//前破壞電磁閥
F_TRIG_2(CLK:=SOL_S8_VacuumF);
interlockback[3]:=TRUE;
interlockout[3]:=TRUE;
(*SET*)
IF ((F_TRIG_2.Q AND NOT(solstatus[3]))) AND interlockout[3] THEN
	SOL_S8_BreakF:=TRUE;
END_IF;
(*RESET*)
TON_BreakF(In:=SOL_S8_BreakF, PT:=t#500ms);
IF ((TON_BreakF.Q AND (solstatus[3]))) AND interlockback[3] THEN
	SOL_S8_BreakF:=FALSE;
END_IF;
(*STATUS*)
solstatus[3]:=SOL_S8_BreakF;

//後吸取電磁閥
R_TRIG_1[4](CLK:=HMIPB_SOL_S8_VacuumR AND NOT(AutoStatus));
interlockback[4]:=TRUE;
interlockout[4]:=TRUE;
(*SET*)
IF ((R_TRIG_1[4].Q AND NOT(solstatus[4])) OR Autoflow=3) AND interlockout[4] THEN
	SOL_S8_VacuumR:=TRUE;
END_IF;
(*RESET*)
IF ((R_TRIG_1[4].Q AND (solstatus[4])) OR Autoflow=7 OR Initflow=7 OR ErrorStatus[8]) AND interlockback[4] THEN
	SOL_S8_VacuumR:=FALSE;
END_IF;
(*STATUS*)
solstatus[4]:=SOL_S8_VacuumR;

//後破壞電磁閥
F_TRIG_3(CLK:=SOL_S8_VacuumR);
interlockback[5]:=TRUE;
interlockout[5]:=TRUE;
(*SET*)
IF ((F_TRIG_3.Q AND NOT(solstatus[5]))) AND interlockout[5] THEN
	SOL_S8_BreakR:=TRUE;
END_IF;
(*RESET*)
TON_BreakR(In:=SOL_S8_BreakR, PT:=t#500ms);
IF ((TON_BreakR.Q AND (solstatus[5]))) AND interlockback[5] THEN
	SOL_S8_BreakR:=FALSE;
END_IF;
(*STATUS*)
solstatus[5]:=SOL_S8_BreakR;
(*************************************************************************
程序名稱:第8站卡子RESET流程
作者:蔡相偉
版本,日期,版本資訊:
1.0.0		2017/11/22		初始版本

PowerOn=0
Idle=1
夾取回=7
上下回=8
移位回=9
*************************************************************************)
//PowerOn=0
IF NOT(SystemReadyStatus) THEN
	Initflow:=0;
END_IF;

//Idle=1
IF Initflow=0 AND SystemReadyStatus THEN
	Initflow:=1;
END_IF;

IF Initflow=9 AND LS_S8_MoveBack THEN
	Initflow:=1;
END_IF;

//夾取回=7
F_TRIG_1(CLK:= ErrorStatus[8] OR Error_PB_Estop);
IF Initflow=1 AND (F_TRIG_1.Q OR Manual2AutoFlag) THEN
	Initflow:=7;
END_IF;

//上下回=8
IF Initflow=7 AND NOT(SOL_S8_VacuumF) AND NOT(SNR_S8_VacuumF) AND NOT(SOL_S8_VacuumR) AND NOT(SNR_S8_VacuumR) THEN
	Initflow:=8;
END_IF;

//移位回=9
IF Initflow=8 AND LS_S8_UpDownBack THEN
	Initflow:=9;
END_IF;

//*************************************************************************
//Cycle Time
//*************************************************************************
TON_CT(In:=AutoFlow>1, PT:=t#500s);
IF Autoflow>1 THEN
CycleTime[8]:=LINT_TO_REAL(TimeToNanoSec( TON_CT.ET))/1000000000.0;
END_IF;
END_PROGRAM

PROGRAM prStation8_CCD
VAR
    Autoflow : INT;
    R_TRIG_1 : R_TRIG;
    F_TRIG_1 : F_TRIG;
END_VAR
VAR_EXTERNAL
    SystemReadyStatus : BOOL;
    AutoStatus : BOOL;
    HMIPB_OMRON_FQ2_Trig : BOOL;
    OMRON_FQ2_Trig : BOOL;
    OMRON_FQ2_IN0 : BOOL;
    OMRON_FQ2_IN1 : BOOL;
    OMRON_FQ2_IN2 : BOOL;
    OMRON_FQ2_IN3 : BOOL;
    OMRON_FQ2_IN4 : BOOL;
    OMRON_FQ2_IN5 : BOOL;
    CCD_Check_NG : BOOL;
    OMRON_FQ2_Ready : BOOL;
    OMRON_FQ2_NG : BOOL;
    CCDStartFlag : BOOL;
    CCDFinishFlag : BOOL;
END_VAR
(*************************************************************************
程序名稱:CCD流程
作者:蔡相偉
版本,日期,版本資訊:
1.0.0	2016/6/3		初始版本,SNR感測到立即拍照
2.0.0	2016/10/11		修改在轉盤站上使用
流程
PowerOn=0
Idle=1
工件到位=5
CCD拍攝中=2
CCD拍攝完成=3
CCD判定資料記錄=4
工件離開=6
*************************************************************************)
//PowerOn=0
IF NOT(SystemReadyStatus AND AutoStatus) THEN
	AutoFlow:=0;
END_IF;

(*Idle=1*)
IF AutoFlow=0 AND SystemReadyStatus AND AutoStatus THEN
	AutoFlow:=1;
END_IF;

IF AutoFlow=6 AND NOT(CCDStartFlag) THEN
	AutoFlow:=1;
END_IF;

(*工件到位=5*)
IF Autoflow=1 AND CCDStartFlag THEN
	Autoflow:=5;
	CCD_Check_NG:=FALSE;
END_IF;

(*CCD拍攝中=2*)
IF AutoFlow=5  AND OMRON_FQ2_Ready THEN
	AutoFlow:=2;
END_IF;

(*CCD拍攝完成=3*)
IF AutoFlow=2 AND NOT(OMRON_FQ2_Ready) THEN
	AutoFlow:=3;
END_IF;

(*CCD判定資料記錄=4*)
IF AutoFlow=3 THEN
	AutoFlow:=4;
END_IF;

(*工件離開=6*)
IF AutoFlow=4 THEN
	IF OMRON_FQ2_NG THEN
		CCD_Check_NG:=TRUE;
	END_IF;
	AutoFlow:=6;
END_IF;
IF Autoflow=6 THEN
	CCDFinishFlag:=TRUE;
ELSE
	CCDFinishFlag:=FALSE;
END_IF;

//****************************************************************************************
(*手動*)
R_TRIG_1(CLK:= HMIPB_OMRON_FQ2_Trig);
IF R_TRIG_1.Q OR AutoFlow=5 THEN
	OMRON_FQ2_Trig:=TRUE;
END_IF;
F_TRIG_1(CLK:= HMIPB_OMRON_FQ2_Trig);
IF F_TRIG_1.Q OR AutoFlow=2 THEN
	OMRON_FQ2_Trig:=FALSE;
END_IF;

(*場景選擇*)
OMRON_FQ2_IN0:=FALSE;
OMRON_FQ2_IN1:=FALSE;
OMRON_FQ2_IN2:=FALSE;
OMRON_FQ2_IN3:=FALSE;
OMRON_FQ2_IN4:=FALSE;
OMRON_FQ2_IN5:=FALSE;
END_PROGRAM

PROGRAM prStation8_ChangeJig
VAR
    interlockback : ARRAY[0..5] OF BOOL;
    interlockout : ARRAY[0..5] OF BOOL;
    R_TRIG_1 : ARRAY[0..5] OF R_TRIG;
    solstatus : ARRAY[0..5] OF BOOL;
    Autoflow : INT;
    Initflow : INT;
    F_TRIG_1 : F_TRIG;
    Rtrig_test : R_TRIG;
    TON1 : TON;
END_VAR
VAR_EXTERNAL
    HMIPB_SOL_S8_Fix : BOOL;
    AutoStatus : BOOL;
    SOL_S8_Fix : BOOL;
    HMIPB_SOL_S8_FixMove : BOOL;
    SOL_S8_FixMove : BOOL;
    HMIPB_SOL_S8_Turn : BOOL;
    SOL_S8_Turn : BOOL;
    HMIPB_SOL_S8_Clip : BOOL;
    SOL_S8_Clip : BOOL;
    SystemReadyStatus : BOOL;
    CCDStartFlag : BOOL;
    CCD_Check_NG : BOOL;
    S8_ChangeJigStartFlag : BOOL;
    LS_S8_FixMoveOut : BOOL;
    ErrorStatus_S8_Fix : BOOL;
    LS_S8_ClipOut : BOOL;
    LS_S8_FixOut : BOOL;
    LS_S8_TurnOut : BOOL;
    LS_S8_FixBack : BOOL;
    LS_S8_ClipBack : BOOL;
    LS_S8_FixMoveBack : BOOL;
    LS_S8_TurnBack : BOOL;
    LS_S8_MoveBack : BOOL;
    ErrorStatus : ARRAY[0..19] OF BOOL;
    Error_PB_EStop : BOOL;
    Manual2AutoFlag : BOOL;
    StepMode : BOOL;
    LS_S8_UpDownBack : BOOL;
    SOL_S8_UpDown : BOOL;
END_VAR
(*************************************************************************
程序名稱:換卡子方向流程
作者:蔡相偉
版本,日期,版本資訊:
1.0.0		2017/11/29		初始版本

PowerOn=0
Idle=1
前後出=2
夾取出=3
定位出=4
旋轉出=5
定位回=6
夾取回=7
前後回=8
旋轉回=9
*************************************************************************)
//PowerOn=0
IF NOT(SystemReadyStatus AND AutoStatus AND NOT(ErrorStatus_S8_Fix)) THEN
	AutoFlow:=0;
END_IF;

(*Idle=1*)
IF AutoFlow=0 AND SystemReadyStatus AND AutoStatus AND NOT(ErrorStatus_S8_Fix) THEN
	AutoFlow:=1;
END_IF;

IF AutoFlow=9 AND LS_S8_TurnBack THEN
	AutoFlow:=1;
END_IF;

//前後出=2
IF Autoflow=1 AND S8_ChangeJigStartFlag AND Initflow=1 THEN
	Autoflow:=2;
END_IF;

//夾取出=3
IF Autoflow=2 AND LS_S8_FixMoveOut AND (Rtrig_test.Q OR NOT(StepMode)) THEN
	Autoflow:=3;
END_IF;

//定位出=4
IF Autoflow=3 AND LS_S8_ClipOut AND (Rtrig_test.Q OR NOT(StepMode)) THEN
	Autoflow:=4;
END_IF;

//旋轉出=5
IF Autoflow=4 AND LS_S8_FixOut AND (Rtrig_test.Q OR NOT(StepMode)) THEN
	Autoflow:=5;
END_IF;
TON1(In:=Autoflow=5 AND LS_S8_TurnOut, PT:=t#300ms);
//定位回=6
IF Autoflow=5 AND TON1.Q AND (Rtrig_test.Q OR NOT(StepMode)) THEN
	Autoflow:=6;
	S8_ChangeJigStartFlag:=FALSE;
END_IF;

//夾取回=7
IF Autoflow=6 AND LS_S8_FixBack AND (Rtrig_test.Q OR NOT(StepMode)) THEN
	Autoflow:=7;
END_IF;

//前後回=8
IF Autoflow=7 AND LS_S8_ClipBack AND (Rtrig_test.Q OR NOT(StepMode)) THEN
	Autoflow:=8;
END_IF;

//旋轉回=9
IF Autoflow=8 AND LS_S8_FixMoveBack AND (Rtrig_test.Q OR NOT(StepMode)) THEN
	Autoflow:=9;
END_IF;

//*************************************************************************
//手動
//定位電磁閥
R_TRIG_1[0](CLK:=HMIPB_SOL_S8_Fix AND NOT(AutoStatus));
interlockback[0]:=TRUE;
interlockout[0]:=TRUE;
(*SET*)
IF ((R_TRIG_1[0].Q AND NOT(solstatus[0])) OR Autoflow=4) AND interlockout[0] THEN
	SOL_S8_Fix:=TRUE;
END_IF;
(*RESET*)
IF ((R_TRIG_1[0].Q AND (solstatus[0])) OR Autoflow=6 OR Initflow=6) AND interlockback[0] THEN
	SOL_S8_Fix:=FALSE;
END_IF;
(*STATUS*)
solstatus[0]:=SOL_S8_Fix;

//定位前後電磁閥
R_TRIG_1[1](CLK:=HMIPB_SOL_S8_FixMove AND NOT(AutoStatus));
interlockback[1]:=TRUE;
interlockout[1]:=TRUE;
(*SET*)
IF ((R_TRIG_1[1].Q AND NOT(solstatus[1])) OR Autoflow=2) AND interlockout[1] THEN
	SOL_S8_FixMove:=TRUE;
END_IF;
(*RESET*)
IF ((R_TRIG_1[1].Q AND (solstatus[1])) OR Autoflow=8 OR Initflow=8) AND interlockback[1] THEN
	SOL_S8_FixMove:=FALSE;
END_IF;
(*STATUS*)
solstatus[1]:=SOL_S8_FixMove;

//定位旋轉電磁閥
R_TRIG_1[2](CLK:=HMIPB_SOL_S8_Turn AND NOT(AutoStatus));
interlockback[2]:=(LS_S8_FixOut AND SOL_S8_Fix AND LS_S8_UpDownBack AND NOT(SOL_S8_UpDown)) OR LS_S8_FixMoveBack;
interlockout[2]:=(LS_S8_FixOut AND SOL_S8_Fix AND LS_S8_UpDownBack AND NOT(SOL_S8_UpDown)) OR LS_S8_FixMoveBack;
(*SET*)
IF ((R_TRIG_1[2].Q AND NOT(solstatus[2])) OR Autoflow=5) AND interlockout[2] THEN
	SOL_S8_Turn:=TRUE;
END_IF;
(*RESET*)
IF ((R_TRIG_1[2].Q AND (solstatus[2])) OR Autoflow=9 OR Initflow=9) AND interlockback[2] THEN
	SOL_S8_Turn:=FALSE;
END_IF;
(*STATUS*)
solstatus[2]:=SOL_S8_Turn;

//定位夾持電磁閥
R_TRIG_1[3](CLK:=HMIPB_SOL_S8_Clip AND NOT(AutoStatus));
interlockback[3]:=TRUE;
interlockout[3]:=TRUE;
(*SET*)
IF ((R_TRIG_1[3].Q AND NOT(solstatus[3])) OR Autoflow=3) AND interlockout[3] THEN
	SOL_S8_Clip:=TRUE;
END_IF;
(*RESET*)
IF ((R_TRIG_1[3].Q AND (solstatus[3])) OR Autoflow=7 OR Initflow=7) AND interlockback[3] THEN
	SOL_S8_Clip:=FALSE;
END_IF;
(*STATUS*)
solstatus[3]:=SOL_S8_Clip;
(*************************************************************************
程序名稱:換卡子方向RESET流程
作者:蔡相偉
版本,日期,版本資訊:
1.0.0		2017/11/29		初始版本

PowerOn=0
Idle=1
定位回=6
夾取回=7
前後回=8
旋轉回=9
*************************************************************************)
//PowerOn=0
IF NOT(SystemReadyStatus) THEN
	Initflow:=0;
END_IF;

//Idle=1
IF Initflow=0 AND SystemReadyStatus THEN
	Initflow:=1;
END_IF;

IF Initflow=9 AND LS_S8_TurnBack THEN
	Initflow:=1;
END_IF;

//定位回=6
F_TRIG_1(CLK:= ErrorStatus_S8_Fix);
IF Initflow=1 AND (F_TRIG_1.Q) THEN
	Initflow:=6;
END_IF;

//夾取回=7
IF Initflow=6 AND LS_S8_FixBack THEN
	Initflow:=7;
END_IF;

//前後回=8
IF Initflow=7 AND LS_S8_ClipBack THEN
	Initflow:=8;
END_IF;

//旋轉回=9
IF Initflow=8 AND LS_S8_FixMoveBack THEN
	Initflow:=9;
END_IF;
END_PROGRAM

PROGRAM prStation9
VAR
    interlockback : ARRAY[0..1] OF BOOL;
    interlockout : ARRAY[0..1] OF BOOL;
    solstatus : ARRAY[0..1] OF BOOL;
    R_TRIG_1 : ARRAY[0..1] OF R_TRIG;
    Rtrig_test : R_TRIG;
    F_TRIG_1 : F_TRIG;
    Autoflow : INT;
    Initflow : INT;
    TON1 : TON;
    TON2 : TON;
    TON_CT : TON;
END_VAR
VAR_EXTERNAL
    IndexData : ARRAY[0..19] OF stIndexData;
    DisablePB : ARRAY[0..19] OF BOOL;
    SystemReadyStatus : BOOL;
    AutoStatus : BOOL;
    ErrorStatus : ARRAY[0..19] OF BOOL;
    Error_PB_EStop : BOOL;
    MachineRunStatus : BOOL;
    SNR_Index : BOOL;
    RY_Index : BOOL;
    Manual2AutoFlag : BOOL;
    TestPB : ARRAY[0..19] OF BOOL;
    SNR_S9_Check : BOOL;
    CycleTime : ARRAY[0..19] OF REAL;
    BatchIndexCount : DINT;
    Error_SNR_S9_Check : BOOL;
    PB_Reset : BOOL;
    HMIPB_PB_Reset : BOOL;
    Error_SNR_S5_Check : BOOL;
    BatchNGCount : DINT;
END_VAR
(*************************************************************************
程序名稱:第9站檢查卡子流程
作者:蔡相偉
版本,日期,版本資訊:
1.0.0		2017/11/22		初始版本

PowerOn=0
Idle=1
檢查開始=2
檢查完成=3
*************************************************************************)
(*************************************************************************
異常碼
急停=1
氣缸=2
檢查NG=3
*************************************************************************)
//*************************************************************************
//本站狀態判斷
IF IndexData[9].OKFlag[9]
	OR IndexData[9].NGFlag[9] THEN
	IndexData[9].FinishFlag[9]:=TRUE;
END_IF;
//前站狀態判斷
IF  NOT(IndexData[9].FinishFlag[8]) OR	IndexData[9].NGFlag[8] THEN
	IndexData[9].NGFlag[9]:=TRUE;
END_IF;
//本站關閉判斷
IF DisablePB[9] AND IndexData[9].FinishFlag[8] AND IndexData[9].OKFlag[8] AND NOT(IndexData[9].NGFlag[8]) THEN
	IndexData[9].OKFlag[9]:=TRUE;
END_IF;

Rtrig_test(CLK:=TestPB[9]);
//PowerOn=0
IF NOT(SystemReadyStatus AND AutoStatus AND NOT(ErrorStatus[9]) AND NOT(Error_PB_EStop)) THEN
	Autoflow:=0;
END_IF;
	//EStop異常碼
	(*IF Error_PB_Estop AND NOT(IndexData[4].FinishFlag[4]) AND IndexData[4].OkFlag[1] THEN
		IndexData[4].NGFlag[4]:=TRUE;
		IndexData[4].ErrorLog[4]:=1;
	END_IF;*)
	//Error異常碼
	(*IF ErrorStatus[4] AND NOT(IndexData[4].FinishFlag[4]) AND IndexData[4].OkFlag[1] THEN
		IndexData[4].NGFlag[4]:=TRUE;
		IndexData[4].ErrorLog[4]:=2;
	END_IF;*)
//Idle=1
IF AutoFlow=0 AND SystemReadyStatus AND AutoStatus AND NOT(ErrorStatus[9]) AND NOT(Error_PB_EStop) THEN
	AutoFlow:=1;
END_IF;

IF Autoflow=3 AND IndexData[9].FinishFlag[9] THEN
	Autoflow:=1;
END_IF;

//檢查開始=2
IF Autoflow=1
	AND AutoStatus
	AND NOT(DisablePB[9])
	AND SNR_Index
	AND NOT(RY_Index)
	AND (MachineRunStatus AND NOT(IndexData[9].FinishFlag[9]) AND IndexData[9].FinishFlag[8] AND IndexData[9].OKFlag[8] AND NOT(IndexData[9].NGFlag[8])
	OR Rtrig_test.Q) THEN
	Autoflow:=2;
	Error_SNR_S9_Check:=FALSE;
END_IF;
TON1(In:=Autoflow=2 AND SNR_S9_Check, PT:=t#500ms);		//OK
TON2(In:=Autoflow=2 AND NOT(TON1.Q), PT:=t#1000ms);		//NG
//檢查完成=3
IF Autoflow=2 AND TON1.Q THEN
	IndexData[9].OKFlag[9]:=TRUE;
	IndexData[9].NGFlag[9]:=FALSE;
	IndexData[9].ErrorLog[9]:=0;
	Autoflow:=3;
END_IF;
IF Autoflow=2 AND TON2.Q THEN
	Error_SNR_S9_Check:=TRUE;
	IndexData[9].OKFlag[9]:=FALSE;
	IndexData[9].NGFlag[9]:=TRUE;
	IndexData[9].ErrorLog[9]:=3;
	BatchIndexCount:=BatchIndexCount-1;
	BatchNGCount:=BatchNGCount+1;
	Autoflow:=3;
END_IF;
IF NOT(SNR_Index) THEN
	Error_SNR_S9_Check:=FALSE;
END_IF;
//*************************************************************************
//Cycle Time
//*************************************************************************
TON_CT(In:=AutoFlow>1, PT:=t#500s);
IF Autoflow>1 THEN
CycleTime[9]:=LINT_TO_REAL(TimeToNanoSec( TON_CT.ET))/1000000000.0;
END_IF;
END_PROGRAM

PROGRAM prStation10
VAR
    interlockback : ARRAY[0..4] OF BOOL;
    interlockout : ARRAY[0..4] OF BOOL;
    solstatus : ARRAY[0..4] OF BOOL;
    R_TRIG_1 : ARRAY[0..4] OF R_TRIG;
    Rtrig_test : R_TRIG;
    F_TRIG_1 : F_TRIG;
    Autoflow : INT;
    Initflow : INT;
    TON1 : TON;
    TON2 : TON;
    TON_CT : TON;
END_VAR
VAR_EXTERNAL
    HMIPB_SOL_S10_MoveBack : BOOL;
    AutoStatus : BOOL;
    SOL_S10_MoveBack : BOOL;
    SOL_S10_MoveOut : BOOL;
    LS_S10_MoveBack : BOOL;
    HMIPB_SOL_S10_MoveOut : BOOL;
    LS_S10_MoveOut : BOOL;
    HMIPB_SOL_S10_UpDown : BOOL;
    SOL_S10_UpDown : BOOL;
    IndexData : ARRAY[0..19] OF stIndexData;
    DisablePB : ARRAY[0..19] OF BOOL;
    TestPB : ARRAY[0..19] OF BOOL;
    SystemReadyStatus : BOOL;
    ErrorStatus : ARRAY[0..19] OF BOOL;
    Error_PB_EStop : BOOL;
    Error_SNR_S10_Feed : BOOL;
    LS_S10_UpDownBack : BOOL;
    MachineRunStatus : BOOL;
    LS_S10_UpDownOut : BOOL;
    SNR_Index : BOOL;
    RY_Index : BOOL;
    Manual2AutoFlag : BOOL;
    YAMAHA_ORG : BOOL;
    SNR_S10_Feed : BOOL;
    FeedStart : ARRAY[0..19] OF BOOL;
    FeedFinish : ARRAY[0..19] OF BOOL;
    ErrorStatus_TH : ARRAY[0..19] OF BOOL;
    LS_S2_UpDownOut : BOOL;
    HMIPB_SOL_S10_ClipF : BOOL;
    SOL_S10_ClipF : BOOL;
    HMIPB_SOL_S10_ClipR : BOOL;
    SOL_S10_ClipR : BOOL;
    HMIPB_SOL_S10_Turn : BOOL;
    SOL_S10_Turn : BOOL;
    LS_S10_THBack : BOOL;
    LS_S10_ClipFBack : BOOL;
    LS_S10_ClipRBack : BOOL;
    LS_S10_TurnBack : BOOL;
    LS_S10_ClipFOut : BOOL;
    LS_S10_ClipROut : BOOL;
    LS_S10_TurnOut : BOOL;
    CycleTime : ARRAY[0..19] OF REAL;
    BatchIndexCount : DINT;
    Error_LS_S10_UpDownOut1 : BOOL;
    StepMode : BOOL;
    BatchNGCount : DINT;
END_VAR
(*************************************************************************
程序名稱:第10站上夾板流程
作者:蔡相偉
版本,日期,版本資訊:
1.0.0		2017/11/22		初始版本

PowerOn=0
Idle=1
上下出=2
夾取出=3
上下回=4
移位出,旋轉出=5
上下出=6
夾取回=7
上下回=8
移位回,旋轉回=9
*************************************************************************)
(*************************************************************************
異常碼
急停=1
氣缸=2
轉子組放入失敗=3
*************************************************************************)
//*************************************************************************
//本站狀態判斷
IF IndexData[10].OKFlag[10]
	OR IndexData[10].NGFlag[10] THEN
	IndexData[10].FinishFlag[10]:=TRUE;
END_IF;
IF  NOT(IndexData[10].FinishFlag[9]) OR	IndexData[10].NGFlag[9] THEN
	IndexData[10].NGFlag[10]:=TRUE;
END_IF;

IF DisablePB[10] AND IndexData[10].FinishFlag[9] AND IndexData[10].OKFlag[9] AND NOT(IndexData[10].NGFlag[9]) THEN
	IndexData[10].OKFlag[10]:=TRUE;
END_IF;

Rtrig_test(CLK:=TestPB[10]);
//PowerOn=0
IF NOT(SystemReadyStatus AND AutoStatus AND NOT(ErrorStatus[10]) AND NOT(Error_PB_EStop)) THEN
	Autoflow:=0;
END_IF;
	//EStop異常碼
	IF Error_PB_Estop AND NOT(IndexData[10].FinishFlag[10]) AND IndexData[10].OkFlag[1] THEN
		IndexData[10].NGFlag[10]:=TRUE;
		IndexData[10].ErrorLog[10]:=1;
		BatchIndexCount:=BatchIndexCount-1;
		BatchNGCount:=BatchNGCount+1;
	END_IF;
	//Error異常碼
	IF ErrorStatus[10] AND NOT(IndexData[10].FinishFlag[10]) AND IndexData[10].OkFlag[1] THEN
		IndexData[10].NGFlag[10]:=TRUE;
		IndexData[10].ErrorLog[10]:=2;
		BatchIndexCount:=BatchIndexCount-1;
		BatchNGCount:=BatchNGCount+1;
	END_IF;
//Idle=1
IF AutoFlow=0 AND SystemReadyStatus AND AutoStatus AND NOT(ErrorStatus[10]) AND NOT(Error_PB_EStop) THEN
	AutoFlow:=1;
END_IF;

IF Autoflow=9 AND LS_S10_MoveBack THEN
	Autoflow:=1;
END_IF;

//上下出=2
IF Autoflow=1
	AND AutoStatus
	AND NOT(DisablePB[10])
	AND LS_S10_THBack
	AND LS_S10_TurnBack
	AND LS_S10_MoveBack
	AND LS_S10_UpDownBack
	AND LS_S10_ClipFBack
	AND LS_S10_ClipRBack
	AND (MachineRunStatus AND NOT(IndexData[10].FinishFlag[10]) AND IndexData[10].FinishFlag[9] AND IndexData[10].OKFlag[9] AND NOT(IndexData[10].NGFlag[9])
	OR Rtrig_test.Q) THEN
	Autoflow:=2;
	Error_LS_S10_UpDownOut1:=FALSE;
END_IF;

//夾取出=3
IF Autoflow=2 AND LS_S10_UpDownOut AND (Rtrig_test.Q OR NOT(StepMode)) THEN
	Autoflow:=3;
END_IF;

//上下回=4
IF Autoflow=3 AND LS_S10_ClipFOut AND LS_S10_ClipROut AND (Rtrig_test.Q OR NOT(StepMode)) THEN
	Autoflow:=4;
END_IF;

//移位出,旋轉出=5
IF Autoflow=4 AND LS_S10_UpDownBack AND (Rtrig_test.Q OR NOT(StepMode)) THEN
	Autoflow:=5;
	FeedStart[10]:=TRUE;
END_IF;
IF FeedFinish[10] THEN
	FeedStart[10]:=FALSE;
END_IF;

//上下出=6
IF Autoflow=5 AND LS_S10_MoveOut AND LS_S10_TurnOut AND (Rtrig_test.Q OR NOT(StepMode)) THEN
	Autoflow:=6;
END_IF;
TON1(In:=Autoflow=6 AND LS_S10_UpDownOut, PT:=t#500ms);		//OK
TON2(In:=Autoflow=6 AND NOT(TON1.Q), PT:=t#2000ms);		//NG

//夾取回=7
IF Autoflow=6 AND TON1.Q AND (Rtrig_test.Q OR NOT(StepMode)) THEN
	IndexData[10].OKFlag[10]:=TRUE;
	IndexData[10].NGFlag[10]:=FALSE;
	IndexData[10].ErrorLog[10]:=0;
	Autoflow:=7;
END_IF;
IF Autoflow=6 AND TON2.Q AND (Rtrig_test.Q OR NOT(StepMode)) THEN
	Error_LS_S10_UpDownOut1:=TRUE;
	IndexData[10].OKFlag[10]:=FALSE;
	IndexData[10].NGFlag[10]:=TRUE;
	IndexData[10].ErrorLog[10]:=3;
	BatchIndexCount:=BatchIndexCount-1;
	BatchNGCount:=BatchNGCount+1;
	Autoflow:=7;
END_IF;

//上下回=8
IF Autoflow=7 AND LS_S10_ClipFBack AND LS_S10_ClipRBack AND (Rtrig_test.Q OR NOT(StepMode)) THEN
	Autoflow:=8;
END_IF;

//移位回,旋轉回=9
IF Autoflow=8 AND LS_S10_UpDownBack AND (Rtrig_test.Q OR NOT(StepMode)) THEN
	Autoflow:=9;
END_IF;
//*************************************************************************
//手動
//移位歸電磁閥
interlockback[0]:=LS_S10_UpDownBack AND NOT(SOL_S10_UpDown);
IF ((HMIPB_SOL_S10_MoveBack AND NOT(AutoStatus)) OR Autoflow=9 OR Initflow=9) AND interlockback[0] THEN
	SOL_S10_MoveBack:=TRUE;
	SOL_S10_MoveOut:=FALSE;
END_IF;
IF LS_S10_MoveBack THEN
	SOL_S10_MoveBack:=FALSE;
END_IF;

//移位出電磁閥
interlockout[0]:=LS_S10_UpDownBack AND NOT(SOL_S10_UpDown);
IF ((HMIPB_SOL_S10_MoveOut AND NOT(AutoStatus)) OR Autoflow=5) AND interlockout[0] THEN
	SOL_S10_MoveBack:=FALSE;
	SOL_S10_MoveOut:=TRUE;
END_IF;
IF LS_S10_MoveOut THEN
	SOL_S10_MoveOut:=FALSE;
END_IF;

//上下電磁閥
R_TRIG_1[1](CLK:=HMIPB_SOL_S10_UpDown AND NOT(AutoStatus));
interlockback[1]:=TRUE;
interlockout[1]:=(LS_S10_MoveBack AND LS_S10_TurnBack AND NOT(SOL_S10_Turn)) OR (LS_S10_MoveOut AND LS_S10_TurnOut AND SOL_S10_Turn);
(*SET*)
IF ((R_TRIG_1[1].Q AND NOT(solstatus[1])) OR Autoflow=2 OR Autoflow=6) AND interlockout[1] THEN
	SOL_S10_UpDown:=TRUE;
END_IF;
(*RESET*)
IF ((R_TRIG_1[1].Q AND (solstatus[1])) OR Autoflow=4 OR Autoflow=8 OR Initflow=8) AND interlockback[1] THEN
	SOL_S10_UpDown:=FALSE;
END_IF;
(*STATUS*)
solstatus[1]:=SOL_S10_UpDown;

//前夾持電磁閥
R_TRIG_1[2](CLK:=HMIPB_SOL_S10_ClipF AND NOT(AutoStatus));
interlockback[2]:=TRUE;
interlockout[2]:=TRUE;
(*SET*)
IF ((R_TRIG_1[2].Q AND NOT(solstatus[2])) OR Autoflow=3) AND interlockout[2] THEN
	SOL_S10_ClipF:=TRUE;
END_IF;
(*RESET*)
IF ((R_TRIG_1[2].Q AND (solstatus[2])) OR Autoflow=7 OR Initflow=7) AND interlockback[2] THEN
	SOL_S10_ClipF:=FALSE;
END_IF;
(*STATUS*)
solstatus[2]:=SOL_S10_ClipF;

//後夾持電磁閥
R_TRIG_1[3](CLK:=HMIPB_SOL_S10_ClipR AND NOT(AutoStatus));
interlockback[3]:=TRUE;
interlockout[3]:=TRUE;
(*SET*)
IF ((R_TRIG_1[3].Q AND NOT(solstatus[3])) OR Autoflow=3) AND interlockout[3] THEN
	SOL_S10_ClipR:=TRUE;
END_IF;
(*RESET*)
IF ((R_TRIG_1[3].Q AND (solstatus[3])) OR Autoflow=7 OR Initflow=7) AND interlockback[3] THEN
	SOL_S10_ClipR:=FALSE;
END_IF;
(*STATUS*)
solstatus[3]:=SOL_S10_ClipR;

//旋轉電磁閥
R_TRIG_1[4](CLK:=HMIPB_SOL_S10_Turn AND NOT(AutoStatus));
interlockback[4]:=TRUE;
interlockout[4]:=TRUE;
(*SET*)
IF ((R_TRIG_1[4].Q AND NOT(solstatus[4])) OR Autoflow=5) AND interlockout[4] THEN
	SOL_S10_Turn:=TRUE;
END_IF;
(*RESET*)
IF ((R_TRIG_1[4].Q AND (solstatus[4])) OR Autoflow=9 OR Initflow=9) AND interlockback[4] THEN
	SOL_S10_Turn:=FALSE;
END_IF;
(*STATUS*)
solstatus[4]:=SOL_S10_Turn;
(*************************************************************************
程序名稱:第10站上夾板RESET流程
作者:蔡相偉
版本,日期,版本資訊:
1.0.0		2017/11/22		初始版本

PowerOn=0
Idle=1
夾取回=7
上下回=8
移位回,旋轉回=9
*************************************************************************)
//PowerOn=0
IF NOT(SystemReadyStatus) THEN
	Initflow:=0;
END_IF;

//Idle=1
IF Initflow=0 AND SystemReadyStatus THEN
	Initflow:=1;
END_IF;

IF Initflow=9 AND LS_S10_MoveBack THEN
	Initflow:=1;
END_IF;

//夾取回=7
F_TRIG_1(CLK:= ErrorStatus[10] OR Error_PB_Estop);
IF Initflow=1 AND (F_TRIG_1.Q OR Manual2AutoFlag) THEN
	Initflow:=7;
END_IF;

//上下回=8
IF Initflow=7 AND LS_S10_ClipFBack AND LS_S10_ClipRBack THEN
	Initflow:=8;
END_IF;

//移位回,旋轉回=9
IF Initflow=8 AND LS_S10_UpDownBack THEN
	Initflow:=9;
END_IF;

//*************************************************************************
//Cycle Time
//*************************************************************************
TON_CT(In:=AutoFlow>1, PT:=t#500s);
IF Autoflow>1 THEN
CycleTime[10]:=LINT_TO_REAL(TimeToNanoSec( TON_CT.ET))/1000000000.0;
END_IF;
END_PROGRAM

PROGRAM prStation11
VAR
    interlockback : ARRAY[0..1] OF BOOL;
    interlockout : ARRAY[0..1] OF BOOL;
    solstatus : ARRAY[0..1] OF BOOL;
    R_TRIG_1 : ARRAY[0..1] OF R_TRIG;
    Rtrig_test : R_TRIG;
    F_TRIG_1 : F_TRIG;
    Autoflow : INT;
    Initflow : INT;
    TON1 : TON;
    TON2 : TON;
    TON3 : TON;
    TON_CT : TON;
END_VAR
VAR_EXTERNAL
    IndexData : ARRAY[0..19] OF stIndexData;
    DisablePB : ARRAY[0..19] OF BOOL;
    SystemReadyStatus : BOOL;
    AutoStatus : BOOL;
    ErrorStatus : ARRAY[0..19] OF BOOL;
    Error_PB_EStop : BOOL;
    MachineRunStatus : BOOL;
    SNR_Index : BOOL;
    RY_Index : BOOL;
    Manual2AutoFlag : BOOL;
    TestPB : ARRAY[0..19] OF BOOL;
    HMIPB_SOL_S11_UpDown : BOOL;
    SOL_S11_UpDown : BOOL;
    HMISV_S11_StandarValue : INT;
    HMIPV_S11_CurrentValue : INT;
    HMISV_S11_MaxValue : INT;
    HMISV_S11_PValue : INT;
    HMISV_S11_MinValue : INT;
    HMISV_S11_NValue : INT;
    HMIPB_S11_StandarValueSet : BOOL;
    LS_S11_UpDownBack : BOOL;
    LS_S11_UpDownOut : BOOL;
    CycleTime : ARRAY[0..19] OF REAL;
    BatchIndexCount : DINT;
    Error_LS_S11_UpDownOut1 : BOOL;
    StepMode : BOOL;
    HMIPV_S11_ADValue : INT;
    Error_SNR_S5_Check : BOOL;
    BatchNGCount : DINT;
END_VAR
(*************************************************************************
程序名稱:第11站檢查上夾板流程
作者:蔡相偉
版本,日期,版本資訊:
1.0.0		2017/11/28		初始版本

PowerOn=0
Idle=1
上下出=2
檢查開始=3
上下回=4
*************************************************************************)
(*************************************************************************
異常碼
急停=1
氣缸=2
檢查NG=3
*************************************************************************)
//*************************************************************************
//本站狀態判斷
IF IndexData[11].OKFlag[11]
	OR IndexData[11].NGFlag[11] THEN
	IndexData[11].FinishFlag[11]:=TRUE;
END_IF;
//前站狀態判斷
IF  NOT(IndexData[11].FinishFlag[10]) OR	IndexData[11].NGFlag[10] THEN
	IndexData[11].NGFlag[11]:=TRUE;
END_IF;
//本站關閉判斷
IF DisablePB[11] AND IndexData[11].FinishFlag[10] AND IndexData[11].OKFlag[10] AND NOT(IndexData[11].NGFlag[10]) THEN
	IndexData[11].OKFlag[11]:=TRUE;
END_IF;

Rtrig_test(CLK:=TestPB[11]);
//PowerOn=0
IF NOT(SystemReadyStatus AND AutoStatus AND NOT(ErrorStatus[11]) AND NOT(Error_PB_EStop)) THEN
	Autoflow:=0;
END_IF;
	//EStop異常碼
	IF Error_PB_Estop AND NOT(IndexData[11].FinishFlag[11]) AND IndexData[11].OkFlag[1] THEN
		IndexData[11].NGFlag[11]:=TRUE;
		IndexData[11].ErrorLog[11]:=1;
		BatchIndexCount:=BatchIndexCount-1;
		BatchNGCount:=BatchNGCount+1;
	END_IF;
	//Error異常碼
	IF ErrorStatus[11] AND NOT(IndexData[11].FinishFlag[11]) AND IndexData[11].OkFlag[1] THEN
		IndexData[11].NGFlag[11]:=TRUE;
		IndexData[11].ErrorLog[11]:=2;
		BatchIndexCount:=BatchIndexCount-1;
		BatchNGCount:=BatchNGCount+1;
	END_IF;
//Idle=1
IF AutoFlow=0 AND SystemReadyStatus AND AutoStatus AND NOT(ErrorStatus[11]) AND NOT(Error_PB_EStop) THEN
	AutoFlow:=1;
END_IF;

IF Autoflow=4 AND LS_S11_UpDownBack THEN
	Autoflow:=1;
END_IF;

//上下出=2
IF Autoflow=1
	AND AutoStatus
	AND NOT(DisablePB[11])
	AND LS_S11_UpDownBack
	AND NOT(SOL_S11_UpDown)
	AND (MachineRunStatus AND NOT(IndexData[11].FinishFlag[11]) AND IndexData[11].FinishFlag[10] AND IndexData[11].OKFlag[10] AND NOT(IndexData[11].NGFlag[10])
	OR Rtrig_test.Q) THEN
	Autoflow:=2;
	Error_LS_S11_UpDownOut1:=FALSE;
END_IF;
TON1(In:=Autoflow=2 AND LS_S11_UpDownOut, PT:=t#1000ms);
TON3(In:=Autoflow=2 AND NOT(LS_S11_UpDownOut), PT:=t#1000ms);
IF TON3.Q THEN		//NG
	Error_LS_S11_UpDownOut1:=TRUE;
	IndexData[11].OKFlag[11]:=FALSE;
	IndexData[11].NGFlag[11]:=TRUE;
	IndexData[11].ErrorLog[11]:=3;
END_IF;
//檢查開始=3
IF Autoflow=2 AND TON1.Q THEN
	Autoflow:=3;
END_IF;
IF Autoflow=3 AND HMIPV_S11_CurrentValue<=HMISV_S11_MaxValue AND HMIPV_S11_CurrentValue>=HMISV_S11_MinValue THEN		//OK
	IndexData[11].OKFlag[11]:=TRUE;
	IndexData[11].NGFlag[11]:=FALSE;
	IndexData[11].ErrorLog[11]:=0;
END_IF;
IF Autoflow=3 AND (HMIPV_S11_CurrentValue>HMISV_S11_MaxValue OR HMIPV_S11_CurrentValue<HMISV_S11_MinValue) THEN		//NG
	Error_LS_S11_UpDownOut1:=TRUE;
	IndexData[11].OKFlag[11]:=FALSE;
	IndexData[11].NGFlag[11]:=TRUE;
	IndexData[11].ErrorLog[11]:=3;
END_IF;
IF NOT(SNR_Index) THEN
	Error_LS_S11_UpDownOut1:=FALSE;
END_IF;
TON2(In:=Autoflow=3 AND IndexData[11].FinishFlag[11], PT:=t#1000ms);
//上下回=4
IF Autoflow=3 AND TON2.Q AND (Rtrig_test.Q OR NOT(StepMode)) THEN
	Autoflow:=4;
	IF IndexData[11].NGFlag[11] THEN
		BatchIndexCount:=BatchIndexCount-1;
		BatchNGCount:=BatchNGCount+1;
	END_IF;
END_IF;
IF Autoflow=2 AND TON3.Q THEN
	Autoflow:=4;
END_IF;
//*************************************************************************
//手動
//上下電磁閥
R_TRIG_1[0](CLK:=HMIPB_SOL_S11_UpDown AND NOT(AutoStatus));
interlockback[0]:=TRUE;
interlockout[0]:=SNR_Index AND NOT(RY_Index);
(*SET*)
IF ((R_TRIG_1[0].Q AND NOT(solstatus[0])) OR Autoflow=2) AND interlockout[0] THEN
	SOL_S11_UpDown:=TRUE;
END_IF;
(*RESET*)
IF ((R_TRIG_1[0].Q AND (solstatus[0])) OR Autoflow=4 OR Initflow=4) AND interlockback[0] THEN
	SOL_S11_UpDown:=FALSE;
END_IF;
(*STATUS*)
solstatus[0]:=SOL_S11_UpDown;

//人機顯示值
HMIPV_S11_CurrentValue:=REAL_TO_INT(INT_TO_REAL(HMIPV_S11_ADValue)/3.33);
//標準值設定
IF HMIPB_S11_StandarValueSet THEN
	HMISV_S11_StandarValue:=HMIPV_S11_CurrentValue;
END_IF;

HMISV_S11_MaxValue:=HMISV_S11_StandarValue+HMISV_S11_PValue;	//最大值
HMISV_S11_MinValue:=HMISV_S11_StandarValue-HMISV_S11_NValue;	//最小值

(*************************************************************************
程序名稱:第11站檢查上夾板RESET流程
作者:蔡相偉
版本,日期,版本資訊:
1.0.0		2017/11/22		初始版本

PowerOn=0
Idle=1
上下回=4
*************************************************************************)
//PowerOn=0
IF NOT(SystemReadyStatus) THEN
	Initflow:=0;
END_IF;

//Idle=1
IF Initflow=0 AND SystemReadyStatus THEN
	Initflow:=1;
END_IF;

IF Initflow=4 AND LS_S11_UpDownBack THEN
	Initflow:=1;
END_IF;

//上下回=4
F_TRIG_1(CLK:= ErrorStatus[11] OR Error_PB_Estop);
IF Initflow=1 AND (F_TRIG_1.Q OR Manual2AutoFlag) THEN
	Initflow:=4;
END_IF;

//*************************************************************************
//Cycle Time
//*************************************************************************
TON_CT(In:=AutoFlow>1, PT:=t#500s);
IF Autoflow>1 THEN
CycleTime[11]:=LINT_TO_REAL(TimeToNanoSec( TON_CT.ET))/1000000000.0;
END_IF;
END_PROGRAM

PROGRAM prStation13
VAR
    interlockback : ARRAY[0..1] OF BOOL;
    interlockout : ARRAY[0..1] OF BOOL;
    solstatus : ARRAY[0..1] OF BOOL;
    R_TRIG_1 : ARRAY[0..1] OF R_TRIG;
    Rtrig_test : R_TRIG;
    F_TRIG_1 : F_TRIG;
    Autoflow : INT;
    Initflow : INT;
    TON1 : TON;
    TON2 : TON;
    tPressTime : TIME;
    TON_CT : TON;
END_VAR
VAR_EXTERNAL
    IndexData : ARRAY[0..19] OF stIndexData;
    DisablePB : ARRAY[0..19] OF BOOL;
    SystemReadyStatus : BOOL;
    AutoStatus : BOOL;
    ErrorStatus : ARRAY[0..19] OF BOOL;
    Error_PB_EStop : BOOL;
    LS_S13_UpDownBack : BOOL;
    MachineRunStatus : BOOL;
    LS_S13_UpDownOut : BOOL;
    HMIPB_SOL_S13_UpDown : BOOL;
    SNR_Index : BOOL;
    RY_Index : BOOL;
    SOL_S13_UpDown : BOOL;
    Manual2AutoFlag : BOOL;
    TestPB : ARRAY[0..19] OF BOOL;
    LS_S13_TempHighWarring : BOOL;
    LS_S13_TempLowWarring : BOOL;
    Error_LS_S13_TempHighWarring : BOOL;
    Error_LS_S13_TempLowWarring : BOOL;
    HMISV_S13_PressTime : DINT;
    CycleTime : ARRAY[0..19] OF REAL;
    BatchIndexCount : DINT;
    Error_LS_S11_UpDownOut1 : BOOL;
    Error_LS_S13_UpDownOut1 : BOOL;
    StepMode : BOOL;
    BatchNGCount : DINT;
END_VAR
(*************************************************************************
程序名稱:第13站壓合流程
作者:蔡相偉
版本,日期,版本資訊:
1.0.0		2017/11/22		初始版本

PowerOn=0
Idle=1
上下出=2
檢查開始=3
上下回=4
*************************************************************************)
(*************************************************************************
異常碼
急停=1
氣缸=2
檢查NG=3
*************************************************************************)
//*************************************************************************
//本站狀態判斷
IF IndexData[13].OKFlag[13]
	OR IndexData[13].NGFlag[13] THEN
	IndexData[13].FinishFlag[13]:=TRUE;
END_IF;
//前站狀態判斷
IF  NOT(IndexData[13].FinishFlag[11]) OR	IndexData[13].NGFlag[11] THEN
	IndexData[13].NGFlag[13]:=TRUE;
END_IF;
//本站關閉判斷
IF DisablePB[13] AND IndexData[13].FinishFlag[11] AND IndexData[13].OKFlag[11] AND NOT(IndexData[13].NGFlag[11]) THEN
	IndexData[13].OKFlag[13]:=TRUE;
END_IF;

Rtrig_test(CLK:=TestPB[13]);
//PowerOn=0
IF NOT(SystemReadyStatus AND AutoStatus AND NOT(ErrorStatus[13]) AND NOT(Error_PB_EStop)) THEN
	Autoflow:=0;
END_IF;
	//EStop異常碼
	IF Error_PB_Estop AND NOT(IndexData[13].FinishFlag[13]) AND IndexData[13].OkFlag[1] THEN
		IndexData[13].NGFlag[13]:=TRUE;
		IndexData[13].ErrorLog[13]:=1;
		BatchIndexCount:=BatchIndexCount-1;
		BatchNGCount:=BatchNGCount+1;
	END_IF;
	//Error異常碼
	IF ErrorStatus[13] AND NOT(IndexData[13].FinishFlag[13]) AND IndexData[13].OkFlag[1] THEN
		IndexData[13].NGFlag[13]:=TRUE;
		IndexData[13].ErrorLog[13]:=2;
		BatchIndexCount:=BatchIndexCount-1;
		BatchNGCount:=BatchNGCount+1;
	END_IF;
//Idle=1
IF AutoFlow=0 AND SystemReadyStatus AND AutoStatus AND NOT(ErrorStatus[13]) AND NOT(Error_PB_EStop) THEN
	AutoFlow:=1;
END_IF;

IF Autoflow=4 AND LS_S13_UpDownBack THEN
	Autoflow:=1;
END_IF;

//上下出=2
IF Autoflow=1
	AND AutoStatus
	AND NOT(DisablePB[13])
	AND LS_S13_UpDownBack
	AND NOT(SOL_S13_UpDown)
	AND NOT(Error_LS_S13_TempHighWarring)
	AND NOT(Error_LS_S13_TempLowWarring)
	AND (MachineRunStatus AND NOT(IndexData[13].FinishFlag[13]) AND IndexData[13].FinishFlag[11] AND IndexData[13].OKFlag[11] AND NOT(IndexData[13].NGFlag[11])
	OR Rtrig_test.Q) THEN
	Autoflow:=2;
	Error_LS_S13_UpDownOut1:=FALSE;
END_IF;

//檢查開始=3
IF Autoflow=2 AND NOT(LS_S13_UpDownBack) THEN
	Autoflow:=3;
END_IF;
tPressTime:=NanoSecToTime(HMISV_S13_PressTime*100000000);	//Define
TON1(In:=Autoflow=3 AND LS_S13_UpDownOut, PT:=tPressTime);		//OK
TON2(In:=Autoflow=3 AND NOT(TON1.Q), PT:=t#3s);		//NG
//上下回=4
IF Autoflow=3 AND TON1.Q AND (Rtrig_test.Q OR NOT(StepMode)) THEN
	IndexData[13].OKFlag[13]:=TRUE;
	IndexData[13].NGFlag[13]:=FALSE;
	IndexData[13].ErrorLog[13]:=0;
	Autoflow:=4;
END_IF;

IF Autoflow=3 AND TON2.Q AND (Rtrig_test.Q OR NOT(StepMode)) THEN
	Error_LS_S13_UpDownOut1:=TRUE;
	IndexData[13].OKFlag[13]:=FALSE;
	IndexData[13].NGFlag[13]:=TRUE;
	IndexData[13].ErrorLog[13]:=3;
	BatchIndexCount:=BatchIndexCount-1;
	BatchNGCount:=BatchNGCount+1;
	Autoflow:=4;
END_IF;
IF NOT(SNR_Index) THEN
	Error_LS_S13_UpDownOut1:=FALSE;
END_IF;
//*************************************************************************
//手動
//上下電磁閥
R_TRIG_1[0](CLK:=HMIPB_SOL_S13_UpDown AND NOT(AutoStatus));
interlockback[0]:=TRUE;
interlockout[0]:=SNR_Index AND NOT(RY_Index);
(*SET*)
IF ((R_TRIG_1[0].Q AND NOT(solstatus[0])) OR Autoflow=2) AND interlockout[0] THEN
	SOL_S13_UpDown:=TRUE;
END_IF;
(*RESET*)
IF ((R_TRIG_1[0].Q AND (solstatus[0])) OR Autoflow=4 OR Initflow=4) AND interlockback[0] THEN
	SOL_S13_UpDown:=FALSE;
END_IF;
(*STATUS*)
solstatus[0]:=SOL_S13_UpDown;
(*************************************************************************
程序名稱:第13站壓合RESET流程
作者:蔡相偉
版本,日期,版本資訊:
1.0.0		2017/11/22		初始版本

PowerOn=0
Idle=1
上下回=4
*************************************************************************)
//PowerOn=0
IF NOT(SystemReadyStatus) THEN
	Initflow:=0;
END_IF;

//Idle=1
IF Initflow=0 AND SystemReadyStatus THEN
	Initflow:=1;
END_IF;

IF Initflow=4 AND LS_S13_UpDownBack THEN
	Initflow:=1;
END_IF;

//上下回=4
F_TRIG_1(CLK:= ErrorStatus[13] OR Error_PB_Estop);
IF Initflow=1 AND (F_TRIG_1.Q OR Manual2AutoFlag) THEN
	Initflow:=4;
END_IF;

//*************************************************************************
//Cycle Time
//*************************************************************************
TON_CT(In:=AutoFlow>1, PT:=t#500s);
IF Autoflow>1 THEN
CycleTime[13]:=LINT_TO_REAL(TimeToNanoSec( TON_CT.ET))/1000000000.0;
END_IF;
END_PROGRAM

PROGRAM prStation15
VAR
    interlockback : ARRAY[0..1] OF BOOL;
    interlockout : ARRAY[0..1] OF BOOL;
    solstatus : ARRAY[0..1] OF BOOL;
    R_TRIG_1 : ARRAY[0..1] OF R_TRIG;
    Rtrig_test : R_TRIG;
    F_TRIG_1 : F_TRIG;
    Autoflow : INT;
    Initflow : INT;
    TON1 : TON;
    TON2 : TON;
    TON_CT : TON;
    TON3 : TON;
END_VAR
VAR_EXTERNAL
    IndexData : ARRAY[0..19] OF stIndexData;
    DisablePB : ARRAY[0..19] OF BOOL;
    SystemReadyStatus : BOOL;
    AutoStatus : BOOL;
    ErrorStatus : ARRAY[0..19] OF BOOL;
    Error_PB_EStop : BOOL;
    MachineRunStatus : BOOL;
    SNR_Index : BOOL;
    RY_Index : BOOL;
    Manual2AutoFlag : BOOL;
    TestPB : ARRAY[0..19] OF BOOL;
    HMIPB_SOL_S15_UpDown : BOOL;
    SOL_S15_UpDown : BOOL;
    HMISV_S15_StandarValue : INT;
    HMIPV_S15_CurrentValue : INT;
    HMISV_S15_MaxValue : INT;
    HMISV_S15_PValue : INT;
    HMISV_S15_MinValue : INT;
    HMISV_S15_NValue : INT;
    HMIPB_S15_StandarValueSet : BOOL;
    LS_S15_UpDownBack : BOOL;
    LS_S15_UpDownOut : BOOL;
    CycleTime : ARRAY[0..19] OF REAL;
    BatchIndexCount : DINT;
    Error_LS_S13_UpDownOut1 : BOOL;
    Error_LS_S15_UpDownOut1 : BOOL;
    StepMode : BOOL;
    HMIPV_S11_CurrentValue : INT;
    HMIPV_S11_ADValue : INT;
    HMIPV_S15_ADValue : INT;
    LS_S11_UpDownOut : BOOL;
    Error_LS_S11_UpDownOut1 : BOOL;
    BatchNGCount : DINT;
END_VAR
(*************************************************************************
程序名稱:第15站檢查壓合流程
作者:蔡相偉
版本,日期,版本資訊:
1.0.0		2017/11/28		初始版本

PowerOn=0
Idle=1
上下出=2
檢查開始=3
上下回=4
*************************************************************************)
(*************************************************************************
異常碼
急停=1
氣缸=2
檢查NG=3
*************************************************************************)
//*************************************************************************
//本站狀態判斷
IF IndexData[15].OKFlag[15]
	OR IndexData[15].NGFlag[15] THEN
	IndexData[15].FinishFlag[15]:=TRUE;
END_IF;
//前站狀態判斷
IF NOT(IndexData[15].FinishFlag[13]) OR 	IndexData[15].NGFlag[13] THEN
	IndexData[15].NGFlag[15]:=TRUE;
END_IF;
//本站關閉判斷
IF DisablePB[15] AND IndexData[15].FinishFlag[13] AND IndexData[15].OKFlag[13] AND NOT(IndexData[15].NGFlag[13]) THEN
	IndexData[15].OKFlag[15]:=TRUE;
END_IF;

Rtrig_test(CLK:=TestPB[15]);
//PowerOn=0
IF NOT(SystemReadyStatus AND AutoStatus AND NOT(ErrorStatus[15]) AND NOT(Error_PB_EStop)) THEN
	Autoflow:=0;
END_IF;
	//EStop異常碼
	IF Error_PB_Estop AND NOT(IndexData[15].FinishFlag[15]) AND IndexData[15].OkFlag[1] THEN
		IndexData[15].NGFlag[15]:=TRUE;
		IndexData[15].ErrorLog[15]:=1;
		BatchIndexCount:=BatchIndexCount-1;
		BatchNGCount:=BatchNGCount+1;
	END_IF;
	//Error異常碼
	IF ErrorStatus[15] AND NOT(IndexData[15].FinishFlag[15]) AND IndexData[15].OkFlag[1] THEN
		IndexData[15].NGFlag[15]:=TRUE;
		IndexData[15].ErrorLog[15]:=2;
		BatchIndexCount:=BatchIndexCount-1;
		BatchNGCount:=BatchNGCount+1;
	END_IF;
//Idle=1
IF AutoFlow=0 AND SystemReadyStatus AND AutoStatus AND NOT(ErrorStatus[15]) AND NOT(Error_PB_EStop) THEN
	AutoFlow:=1;
END_IF;

IF Autoflow=4 AND LS_S15_UpDownBack THEN
	Autoflow:=1;
END_IF;

//上下出=2
IF Autoflow=1
	AND AutoStatus
	AND NOT(DisablePB[15])
	AND LS_S15_UpDownBack
	AND NOT(SOL_S15_UpDown)
	AND (MachineRunStatus AND NOT(IndexData[15].FinishFlag[15]) AND IndexData[15].FinishFlag[13] AND IndexData[15].OKFlag[13] AND NOT(IndexData[15].NGFlag[13])
	OR Rtrig_test.Q) THEN
	Autoflow:=2;
	Error_LS_S15_UpDownOut1:=FALSE;
END_IF;
TON1(In:=Autoflow=2 AND LS_S15_UpDownOut, PT:=t#1000ms);
TON3(In:=Autoflow=2 AND NOT(LS_S15_UpDownOut), PT:=t#1000ms);
IF TON3.Q THEN		//NG
	Error_LS_S15_UpDownOut1:=TRUE;
	IndexData[15].OKFlag[15]:=FALSE;
	IndexData[15].NGFlag[15]:=TRUE;
	IndexData[15].ErrorLog[15]:=3;
END_IF;
//檢查開始=3
IF Autoflow=2 AND TON1.Q THEN
	Autoflow:=3;
END_IF;
IF Autoflow=3 AND NOT(IndexData[15].FinishFlag[15]) AND HMIPV_S15_CurrentValue<=HMISV_S15_MaxValue AND HMIPV_S15_CurrentValue>=HMISV_S15_MinValue THEN		//OK
	IndexData[15].OKFlag[15]:=TRUE;
	IndexData[15].NGFlag[15]:=FALSE;
	IndexData[15].ErrorLog[15]:=0;
END_IF;
IF Autoflow=3 AND NOT(IndexData[15].FinishFlag[15]) AND (HMIPV_S15_CurrentValue>HMISV_S15_MaxValue OR HMIPV_S15_CurrentValue<HMISV_S15_MinValue) THEN		//NG
	Error_LS_S15_UpDownOut1:=TRUE;
	IndexData[15].OKFlag[15]:=FALSE;
	IndexData[15].NGFlag[15]:=TRUE;
	IndexData[15].ErrorLog[15]:=3;
	BatchIndexCount:=BatchIndexCount-1;
	BatchNGCount:=BatchNGCount+1;
END_IF;
IF NOT(SNR_Index) THEN
	Error_LS_S15_UpDownOut1:=FALSE;
END_IF;
TON2(In:=Autoflow=3 AND IndexData[15].FinishFlag[15], PT:=t#1000ms);
//上下回=4
IF Autoflow=3 AND TON2.Q AND (Rtrig_test.Q OR NOT(StepMode)) THEN
	Autoflow:=4;
	IF IndexData[15].NGFlag[15] THEN
		BatchIndexCount:=BatchIndexCount-1;
	END_IF;
END_IF;
IF Autoflow=2 AND TON3.Q THEN
	Autoflow:=4;
END_IF;
//*************************************************************************
//手動
//上下電磁閥
R_TRIG_1[0](CLK:=HMIPB_SOL_S15_UpDown AND NOT(AutoStatus));
interlockback[0]:=TRUE;
interlockout[0]:=SNR_Index AND NOT(RY_Index);
(*SET*)
IF ((R_TRIG_1[0].Q AND NOT(solstatus[0])) OR Autoflow=2) AND interlockout[0] THEN
	SOL_S15_UpDown:=TRUE;
END_IF;
(*RESET*)
IF ((R_TRIG_1[0].Q AND (solstatus[0])) OR Autoflow=4 OR Initflow=4) AND interlockback[0] THEN
	SOL_S15_UpDown:=FALSE;
END_IF;
(*STATUS*)
solstatus[0]:=SOL_S15_UpDown;

//人機顯示值
HMIPV_S15_CurrentValue:=REAL_TO_INT(INT_TO_REAL(HMIPV_S15_ADValue)/3.33);
//標準值設定
IF HMIPB_S15_StandarValueSet THEN
	HMISV_S15_StandarValue:=HMIPV_S15_CurrentValue;
END_IF;

HMISV_S15_MaxValue:=HMISV_S15_StandarValue+HMISV_S15_PValue;	//最大值
HMISV_S15_MinValue:=HMISV_S15_StandarValue-HMISV_S15_NValue;	//最小值

(*************************************************************************
程序名稱:第15站檢查壓合RESET流程
作者:蔡相偉
版本,日期,版本資訊:
1.0.0		2017/11/22		初始版本

PowerOn=0
Idle=1
上下回=4
*************************************************************************)
//PowerOn=0
IF NOT(SystemReadyStatus) THEN
	Initflow:=0;
END_IF;

//Idle=1
IF Initflow=0 AND SystemReadyStatus THEN
	Initflow:=1;
END_IF;

IF Initflow=4 AND LS_S15_UpDownBack THEN
	Initflow:=1;
END_IF;

//上下回=4
F_TRIG_1(CLK:= ErrorStatus[15] OR Error_PB_Estop);
IF Initflow=1 AND (F_TRIG_1.Q OR Manual2AutoFlag) THEN
	Initflow:=4;
END_IF;

//*************************************************************************
//Cycle Time
//*************************************************************************
TON_CT(In:=AutoFlow>1, PT:=t#500s);
IF Autoflow>1 THEN
CycleTime[15]:=LINT_TO_REAL(TimeToNanoSec( TON_CT.ET))/1000000000.0;
END_IF;
END_PROGRAM

PROGRAM prStation16
VAR
    AutoFlow : INT;
    Rtrig_test : R_TRIG;
    Rtrig_test2 : R_TRIG;
    TON_CT : TON;
END_VAR
VAR_EXTERNAL
    IndexData : ARRAY[0..19] OF stIndexData;
    DisablePB : ARRAY[0..19] OF BOOL;
    TestPB : ARRAY[0..19] OF BOOL;
    SystemReadyStatus : BOOL;
    ErrorStatus : ARRAY[0..19] OF BOOL;
    Error_PB_EStop : BOOL;
    AutoStatus : BOOL;
    MachineRunStatus : BOOL;
    HMIPB_YAMAHA_Unload_OKStart : BOOL;
    YAMAHA_Unload_OKStart : BOOL;
    YAMAHA_Unload_Finish : BOOL;
    HMIPB_YAMAHA_Unload_NGStart : BOOL;
    YAMAHA_Unload_NGStart : BOOL;
    CycleTime : ARRAY[0..19] OF REAL;
    BatchOKCount : DINT;
    BatchIndexCount : DINT;
    BatchNGCount : DINT;
    Error_LS_Door : BOOL;
    StepMode : BOOL;
    Error_YAMAHA_S_State_Alarm : BOOL;
END_VAR
(*
程序名稱:第16站下料流程
作者:蔡相偉
版本,日期,版本資訊:
1.0.0		2017/11/21		初始版本
PowerOn=0
Idle=1|--->OK下料開始=10--->OK下料完成=11
		  |--->NG下料開始=20--->NG下料完成=21
*)
//本站狀態判斷
IF IndexData[16].OKFlag[16]
	OR IndexData[16].NGFlag[16] THEN
	IndexData[16].FinishFlag[16]:=TRUE;
END_IF;

//前站狀態判斷
IF NOT(IndexData[16].OKFlag[1]) THEN
	IndexData[16].NGFlag[16]:=TRUE;
END_IF;

(*
//本站關閉判斷
IF DisablePB[1] THEN
	IndexData[1].NGFlag[1]:=TRUE;
END_IF;
*)
//異常放棄
IF (ErrorStatus[16] OR Error_PB_EStop) AND NOT(IndexData[16].FinishFlag[16]) THEN
	IndexData[16].NGFlag[16]:=TRUE;
END_IF;
Rtrig_test(CLK:=HMIPB_YAMAHA_Unload_OKStart);
Rtrig_test2(CLK:=HMIPB_YAMAHA_Unload_NGStart);
//PowerOn=0
IF NOT(SystemReadyStatus AND AutoStatus AND NOT(ErrorStatus[16]) AND NOT(Error_PB_EStop)) THEN
	Autoflow:=0;
END_IF;

//Idle=1
IF AutoFlow=0 AND SystemReadyStatus AND AutoStatus AND NOT(ErrorStatus[16]) AND NOT(Error_PB_EStop) THEN
	AutoFlow:=1;
END_IF;

IF AutoFlow=11 AND NOT(YAMAHA_Unload_OKStart) AND IndexData[16].FinishFlag[16] THEN
	AutoFlow:=1;
END_IF;

IF AutoFlow=21 AND NOT(YAMAHA_Unload_NGStart) AND IndexData[16].FinishFlag[16] THEN
	AutoFlow:=1;
END_IF;

//OK下料開始=10
IF Autoflow=1
	AND AutoStatus
	AND NOT(DisablePB[16])
	AND (MachineRunStatus AND NOT(IndexData[16].FinishFlag[16]) AND IndexData[16].OKFlag[1] AND IndexData[16].FinishFlag[15] AND IndexData[16].OKFlag[15] AND NOT(IndexData[16].NGFlag[15]) OR Rtrig_test.Q) THEN
	Autoflow:=10;
END_IF;
IF AutoFlow=10 THEN
	HMIPB_YAMAHA_Unload_OKStart:=TRUE;
END_IF;
IF YAMAHA_Unload_Finish OR ErrorStatus[16] OR Error_LS_Door THEN
	HMIPB_YAMAHA_Unload_OKStart:=FALSE;
END_IF;

//OK下料完成=11
IF AutoFlow=10 AND (YAMAHA_Unload_Finish) THEN
	BatchOKCount:=BatchOKCount+1;
	BatchIndexCount:=BatchIndexCount-1;
	AutoFlow:=11;
END_IF;
IF AutoFlow=11 THEN
	IndexData[16].OKFlag[16]:=TRUE;
END_IF;

//NG下料開始=20
IF Autoflow=1
	AND AutoStatus
	AND NOT(DisablePB[16])
	AND (MachineRunStatus AND NOT(IndexData[16].FinishFlag[16]) AND IndexData[16].OKFlag[1] AND IndexData[16].FinishFlag[15] AND (IndexData[16].NGFlag[15]) OR Rtrig_test2.Q) THEN
	Autoflow:=20;
END_IF;
IF AutoFlow=20 THEN
	HMIPB_YAMAHA_Unload_NGStart:=TRUE;
END_IF;
IF YAMAHA_Unload_Finish OR ErrorStatus[16] OR Error_LS_Door THEN
	HMIPB_YAMAHA_Unload_NGStart:=FALSE;
END_IF;

//NG下料完成=21
IF AutoFlow=20 AND (YAMAHA_Unload_Finish) THEN
	//BatchNGCount:=BatchNGCount+1;
	AutoFlow:=21;
END_IF;
IF AutoFlow=21 THEN
	IndexData[16].NGFlag[16]:=TRUE;
END_IF;

//*************************************************************************
//Cycle Time
//*************************************************************************
TON_CT(In:=AutoFlow>1, PT:=t#500s);
IF Autoflow>1 THEN
CycleTime[16]:=LINT_TO_REAL(TimeToNanoSec( TON_CT.ET))/1000000000.0;
END_IF;
END_PROGRAM

PROGRAM prFeedAndSupplier
VAR
    Supplier_S6 : fbFull;
    Supplier_S8 : fbFull;
    Supplier_S10 : fbFull;
    Feeder_S6 : fbFeed;
    Feeder_S8 : fbFeed;
    Feeder_S10 : fbFeed;
END_VAR
VAR_EXTERNAL
    SNR_S6_Full : BOOL;
    RY_S6_Full : BOOL;
    Error_SNR_S6_Full : BOOL;
    FullNotExistTime : ARRAY[0..19] OF DINT;
    FullExistTime : ARRAY[0..19] OF DINT;
    FullNotExistErrorTime : ARRAY[0..19] OF DINT;
    SNR_S8_Full : BOOL;
    RY_S8_Full : BOOL;
    Error_SNR_S8_Full : BOOL;
    SNR_S10_Full : BOOL;
    RY_S10_Full : BOOL;
    Error_SNR_S10_Full : BOOL;
    FeedStart : ARRAY[0..19] OF BOOL;
    PB_Reset : BOOL;
    FeedFinish : ARRAY[0..19] OF BOOL;
    Error_LS_S6_THBack : BOOL;
    Error_LS_S6_THOut : BOOL;
    LS_S6_UpDownBack : BOOL;
    SOL_S6_UpDown : BOOL;
    LS_S6_MoveBack : BOOL;
    SNR_S6_Feed : BOOL;
    LS_S6_THBack : BOOL;
    LS_S6_THOut : BOOL;
    HMIPB_SOL_S6_TH : BOOL;
    FeedNotExistTime : ARRAY[0..19] OF DINT;
    FeedExistTime : ARRAY[0..19] OF DINT;
    Error_SNR_S6_Feed : BOOL;
    RY_S6_Feed : BOOL;
    SOL_S6_TH : BOOL;
    Error_LS_S8_THBack : BOOL;
    Error_LS_S8_THOut : BOOL;
    LS_S8_UpDownBack : BOOL;
    SOL_S8_UpDown : BOOL;
    LS_S8_MoveBack : BOOL;
    SNR_S8_Feed : BOOL;
    LS_S8_THBack : BOOL;
    LS_S8_THOut : BOOL;
    HMIPB_SOL_S8_TH : BOOL;
    Error_SNR_S8_Feed : BOOL;
    RY_S8_Feed : BOOL;
    SOL_S8_TH : BOOL;
    Error_LS_S10_THBack : BOOL;
    Error_LS_S10_THOut : BOOL;
    LS_S10_UpDownBack : BOOL;
    SOL_S10_UpDown : BOOL;
    LS_S10_MoveBack : BOOL;
    SNR_S10_Feed : BOOL;
    LS_S10_THBack : BOOL;
    LS_S10_THOut : BOOL;
    HMIPB_SOL_S10_TH : BOOL;
    Error_SNR_S10_Feed : BOOL;
    RY_S10_Feed : BOOL;
    SOL_S10_TH : BOOL;
    Manual2AutoFlag : BOOL;
    HMIPB_PB_Reset : BOOL;
END_VAR
//第6站振動筒
Supplier_S6();
Supplier_S6.bFullSNR:=SNR_S6_Full;
Supplier_S6.iItemNotExistDelayTime:=FullNotExistTime[6];
Supplier_S6.iItemExistTime:=FullExistTime[6];
Supplier_S6.iItemNotExistErrorTime:=FullNotExistErrorTime[6];
RY_S6_Full:=Supplier_S6.bFullRY;
Error_SNR_S6_Full:=Supplier_S6.bFullSNRError;

//第8站振動筒
Supplier_S8();
Supplier_S8.bFullSNR:=SNR_S8_Full;
Supplier_S8.iItemNotExistDelayTime:=FullNotExistTime[8];
Supplier_S8.iItemExistTime:=FullExistTime[8];
Supplier_S8.iItemNotExistErrorTime:=FullNotExistErrorTime[8];
RY_S8_Full:=Supplier_S8.bFullRY;
Error_SNR_S8_Full:=Supplier_S8.bFullSNRError;

//第10站振動筒
Supplier_S10();
Supplier_S10.bFullSNR:=SNR_S10_Full;
Supplier_S10.iItemNotExistDelayTime:=FullNotExistTime[10];
Supplier_S10.iItemExistTime:=FullExistTime[10];
Supplier_S10.iItemNotExistErrorTime:=FullNotExistErrorTime[10];
RY_S10_Full:=Supplier_S10.bFullRY;
Error_SNR_S10_Full:=Supplier_S10.bFullSNRError;

//第6站平送
Feeder_S6();
Feeder_S6.bErrorTHBack:=Error_LS_S6_THBack;
Feeder_S6.bErrorTHOut:=Error_LS_S6_THOut;
Feeder_S6.bFeedStart:=FeedStart[6] OR Manual2AutoFlag;
Feeder_S6.bInterlock_thback:=(LS_S6_UpDownBack AND NOT(SOL_S6_UpDown)) OR NOT(LS_S6_MoveBack);
Feeder_S6.bInterlock_thout:=(LS_S6_UpDownBack AND NOT(SOL_S6_UpDown)) OR NOT(LS_S6_MoveBack);
Feeder_S6.bObjSNR:=SNR_S6_Feed;
Feeder_S6.bReset:=PB_Reset OR HMIPB_PB_Reset;
Feeder_S6.bSupplierRY:=RY_S6_Full;
Feeder_S6.bTHBackLS:=LS_S6_THBack;
Feeder_S6.bTHOutLS:=LS_S6_THOut;
Feeder_S6.bTHPB:=HMIPB_SOL_S6_TH;
Feeder_S6.wNoObjDelayTime:=FeedNotExistTime[6];
Feeder_S6.wObjectExistDelayTime:=FeedExistTime[6];
Error_SNR_S6_Feed :=Feeder_S6.bFeedError;
FeedFinish[6]:= Feeder_S6.bFeedFinish;
RY_S6_Feed:= Feeder_S6.bFeedRY;
SOL_S6_TH:= Feeder_S6.bTHSOL;

//第8站平送
Feeder_S8();
Feeder_S8.bErrorTHBack:=Error_LS_S8_THBack;
Feeder_S8.bErrorTHOut:=Error_LS_S8_THOut;
Feeder_S8.bFeedStart:=FeedStart[8] OR Manual2AutoFlag;
Feeder_S8.bInterlock_thback:=(LS_S8_UpDownBack AND NOT(SOL_S8_UpDown)) OR NOT(LS_S8_MoveBack);
Feeder_S8.bInterlock_thout:=(LS_S8_UpDownBack AND NOT(SOL_S8_UpDown)) OR NOT(LS_S8_MoveBack);
Feeder_S8.bObjSNR:=SNR_S8_Feed;
Feeder_S8.bReset:=PB_Reset OR HMIPB_PB_Reset;
Feeder_S8.bSupplierRY:=RY_S8_Full;
Feeder_S8.bTHBackLS:=LS_S8_THBack;
Feeder_S8.bTHOutLS:=LS_S8_THOut;
Feeder_S8.bTHPB:=HMIPB_SOL_S8_TH;
Feeder_S8.wNoObjDelayTime:=FeedNotExistTime[8];
Feeder_S8.wObjectExistDelayTime:=FeedExistTime[8];
Error_SNR_S8_Feed:=Feeder_S8.bFeedError;
FeedFinish[8]:= Feeder_S8.bFeedFinish;
RY_S8_Feed:= Feeder_S8.bFeedRY;
SOL_S8_TH:= Feeder_S8.bTHSOL;

//第10站平送
Feeder_S10();
Feeder_S10.bErrorTHBack:=Error_LS_S10_THBack;
Feeder_S10.bErrorTHOut:=Error_LS_S10_THOut;
Feeder_S10.bFeedStart:=FeedStart[10] OR Manual2AutoFlag;
Feeder_S10.bInterlock_thback:=(LS_S10_UpDownBack AND NOT(SOL_S10_UpDown)) OR NOT(LS_S10_MoveBack);
Feeder_S10.bInterlock_thout:=(LS_S10_UpDownBack AND NOT(SOL_S10_UpDown)) OR NOT(LS_S10_MoveBack);
Feeder_S10.bObjSNR:=SNR_S10_Feed;
Feeder_S10.bReset:=PB_Reset OR HMIPB_PB_Reset;
Feeder_S10.bSupplierRY:=RY_S10_Full;
Feeder_S10.bTHBackLS:=LS_S10_THBack;
Feeder_S10.bTHOutLS:=LS_S10_THOut;
Feeder_S10.bTHPB:=HMIPB_SOL_S10_TH;
Feeder_S10.wNoObjDelayTime:=FeedNotExistTime[10];
Feeder_S10.wObjectExistDelayTime:=FeedExistTime[10];
Error_SNR_S10_Feed:=Feeder_S10.bFeedError;
FeedFinish[10]:= Feeder_S10.bFeedFinish;
RY_S10_Feed:= Feeder_S10.bFeedRY;
SOL_S10_TH:= Feeder_S10.bTHSOL;
END_PROGRAM

PROGRAM prNGCount
VAR
    R_TRIG1 : ARRAY[0..19] OF R_TRIG;
    iCount : ARRAY[0..19] OF INT;
END_VAR
VAR_EXTERNAL
    IndexData : ARRAY[0..19] OF stIndexData;
    Error_NGCount : ARRAY[0..19] OF BOOL;
    PB_Reset : BOOL;
    HMIPB_PB_Reset : BOOL;
END_VAR
//Over 3 times NG S2
R_TRIG1[0](Clk:=IndexData[2].NGFlag[2]);
IF IndexData[2].OKFlag[1] AND R_TRIG1[0].Q THEN
	iCount[2]:=iCount[2]+1;
END_IF;
IF IndexData[2].OKFlag[2] THEN
	iCount[2]:=0;
END_IF;
IF iCount[2]>=3 THEN
	Error_NGCount[2]:=TRUE;
ELSE
	Error_NGCount[2]:=FALSE;
END_IF;
IF PB_Reset OR HMIPB_PB_Reset THEN
	iCount[2]:=0;
END_IF;

//Over 3 times NG S4
R_TRIG1[1](Clk:=IndexData[4].NGFlag[4]);
IF IndexData[4].OKFlag[1] AND R_TRIG1[1].Q THEN
	iCount[4]:=iCount[4]+1;
END_IF;
IF IndexData[4].OKFlag[4] THEN
	iCount[4]:=0;
END_IF;
IF iCount[4]>=3 THEN
	Error_NGCount[4]:=TRUE;
ELSE
	Error_NGCount[4]:=FALSE;
END_IF;
IF PB_Reset OR HMIPB_PB_Reset THEN
	iCount[4]:=0;
END_IF;

//Over 3 times NG S5
R_TRIG1[2](Clk:=IndexData[5].NGFlag[5]);
IF IndexData[5].OKFlag[1] AND R_TRIG1[2].Q THEN
	iCount[5]:=iCount[5]+1;
END_IF;
IF IndexData[5].OKFlag[5] THEN
	iCount[5]:=0;
END_IF;
IF iCount[5]>=3 THEN
	Error_NGCount[5]:=TRUE;
ELSE
	Error_NGCount[5]:=FALSE;
END_IF;
IF PB_Reset OR HMIPB_PB_Reset THEN
	iCount[5]:=0;
END_IF;

//Over 3 times NG S6
R_TRIG1[3](Clk:=IndexData[6].NGFlag[6]);
IF IndexData[6].OKFlag[1] AND R_TRIG1[3].Q THEN
	iCount[6]:=iCount[6]+1;
END_IF;
IF IndexData[6].OKFlag[6] THEN
	iCount[6]:=0;
END_IF;
IF iCount[6]>=3 THEN
	Error_NGCount[6]:=TRUE;
ELSE
	Error_NGCount[6]:=FALSE;
END_IF;
IF PB_Reset OR HMIPB_PB_Reset THEN
	iCount[6]:=0;
END_IF;

//Over 3 times NG S7
R_TRIG1[4](Clk:=IndexData[7].NGFlag[7]);
IF IndexData[7].OKFlag[1] AND R_TRIG1[4].Q THEN
	iCount[7]:=iCount[7]+1;
END_IF;
IF IndexData[7].OKFlag[7] THEN
	iCount[7]:=0;
END_IF;
IF iCount[7]>=3 THEN
	Error_NGCount[7]:=TRUE;
ELSE
	Error_NGCount[7]:=FALSE;
END_IF;
IF PB_Reset OR HMIPB_PB_Reset THEN
	iCount[7]:=0;
END_IF;

//Over 3 times NG S8
R_TRIG1[5](Clk:=IndexData[8].NGFlag[8]);
IF IndexData[8].OKFlag[1] AND R_TRIG1[5].Q THEN
	iCount[8]:=iCount[8]+1;
END_IF;
IF IndexData[8].OKFlag[8] THEN
	iCount[8]:=0;
END_IF;
IF iCount[8]>=3 THEN
	Error_NGCount[8]:=TRUE;
ELSE
	Error_NGCount[8]:=FALSE;
END_IF;
IF PB_Reset OR HMIPB_PB_Reset THEN
	iCount[8]:=0;
END_IF;

//Over 3 times NG S9
R_TRIG1[6](Clk:=IndexData[9].NGFlag[9]);
IF IndexData[9].OKFlag[1] AND R_TRIG1[6].Q THEN
	iCount[9]:=iCount[9]+1;
END_IF;
IF IndexData[9].OKFlag[9] THEN
	iCount[9]:=0;
END_IF;
IF iCount[9]>=3 THEN
	Error_NGCount[9]:=TRUE;
ELSE
	Error_NGCount[9]:=FALSE;
END_IF;
IF PB_Reset OR HMIPB_PB_Reset THEN
	iCount[9]:=0;
END_IF;

//Over 3 times NG S10
R_TRIG1[7](Clk:=IndexData[10].NGFlag[10]);
IF IndexData[10].OKFlag[1] AND R_TRIG1[7].Q THEN
	iCount[10]:=iCount[10]+1;
END_IF;
IF IndexData[10].OKFlag[10] THEN
	iCount[10]:=0;
END_IF;
IF iCount[10]>=3 THEN
	Error_NGCount[10]:=TRUE;
ELSE
	Error_NGCount[10]:=FALSE;
END_IF;
IF PB_Reset OR HMIPB_PB_Reset THEN
	iCount[10]:=0;
END_IF;

//Over 3 times NG S11
R_TRIG1[8](Clk:=IndexData[11].NGFlag[11]);
IF IndexData[11].OKFlag[1] AND R_TRIG1[8].Q THEN
	iCount[11]:=iCount[11]+1;
END_IF;
IF IndexData[11].OKFlag[11] THEN
	iCount[11]:=0;
END_IF;
IF iCount[11]>=3 THEN
	Error_NGCount[11]:=TRUE;
ELSE
	Error_NGCount[11]:=FALSE;
END_IF;
IF PB_Reset OR HMIPB_PB_Reset THEN
	iCount[11]:=0;
END_IF;

//Over 3 times NG S13
R_TRIG1[9](Clk:=IndexData[13].NGFlag[13]);
IF IndexData[13].OKFlag[1] AND R_TRIG1[9].Q THEN
	iCount[13]:=iCount[13]+1;
END_IF;
IF IndexData[13].OKFlag[13] THEN
	iCount[13]:=0;
END_IF;
IF iCount[13]>=3 THEN
	Error_NGCount[13]:=TRUE;
ELSE
	Error_NGCount[13]:=FALSE;
END_IF;
IF PB_Reset OR HMIPB_PB_Reset THEN
	iCount[13]:=0;
END_IF;

//Over 3 times NG S15
R_TRIG1[10](Clk:=IndexData[15].NGFlag[15]);
IF IndexData[15].OKFlag[1] AND R_TRIG1[10].Q THEN
	iCount[15]:=iCount[15]+1;
END_IF;
IF IndexData[15].OKFlag[15] THEN
	iCount[15]:=0;
END_IF;
IF iCount[15]>=3 THEN
	Error_NGCount[15]:=TRUE;
ELSE
	Error_NGCount[15]:=FALSE;
END_IF;
IF PB_Reset OR HMIPB_PB_Reset THEN
	iCount[15]:=0;
END_IF;
END_PROGRAM

PROGRAM prStation4_feed
VAR
    AutoFlow : INT;
    AutoFlow2 : INT;
    Initflow : INT;
    bStart : BOOL;
    AutoFlow_Ready : BOOL;
    AutoFlow2_Ready : BOOL;
    Unload_Start : BOOL;
    Unload_Finish : BOOL;
    load_Start : BOOL;
    load_Finish : BOOL;
    Error_LS : BOOL;
    MC_MoveAbsolute_X_5_init : MC_MoveAbsolute;
    MC_MoveAbsolute_X_6 : MC_MoveAbsolute;
    MC_MoveAbsolute_Y_6 : MC_MoveAbsolute;
    MC_MoveAbsolute_X_10 : MC_MoveAbsolute;
    MC_MoveAbsolute_X_15 : MC_MoveAbsolute;
    MC_MoveAbsolute_Y_3 : MC_MoveAbsolute;
    MC_MoveAbsolute_Y_7 : MC_MoveAbsolute;
    TON_1 : TON;
    TON_2 : TON;
    TON_3 : TON;
    R_TRIG_1 : R_TRIG;
    R_TRIG_2 : R_TRIG;
    R_TRIG_3 : R_TRIG;
    R_TRIG_4 : R_TRIG;
    R_TRIG_5 : R_TRIG;
    R_TRIG_6 : R_TRIG;
    F_TRIG_1 : F_TRIG;
    Rtrig_test : R_TRIG;
    interlockback : ARRAY[0..2] OF BOOL;
    interlockout : ARRAY[0..2] OF BOOL;
    solStatus : ARRAY[0..2] OF BOOL;
END_VAR
VAR_EXTERNAL
    SystemReadyStatus : BOOL;
    AutoStatus : BOOL;
    Error_PB_EStop : BOOL;
    LS_S4_ClipBack : BOOL;
    LS_S4_UpDownBack : BOOL;
    Ax_X : stAxis;
    LS_S4_Center_ClipBack : BOOL;
    LS_S4_Center_UpDownBack : BOOL;
    Ax_Y : stAxis;
    ServoS4_X_Position : INT;
    ServoS4_Y_Position : INT;
END_VAR
VAR_EXTERNAL CONSTANT
    MC_Axis000 : _sAXIS_REF;
    MC_Axis001 : _sAXIS_REF;
END_VAR
VAR_EXTERNAL
    LS_S4_Center_UpDownOut : BOOL;
    LS_S4_Center_ClipOut : BOOL;
    ServoS4_PutPosition : LREAL;
    ServoS4_StandbyPosition : LREAL;
    ServoS4_UnLoadPosition : LREAL;
    ServoS4_LoadPosition : LREAL;
    HMISV_S4_AbsSpeedX : LREAL;
    HMISV_S4_AbsSpeedY : LREAL;
    ServoS4_X_Table : ARRAY[0..4,0..9] OF LREAL;
    ServoS4_Y_Table : ARRAY[0..4,0..9] OF LREAL;
    StepMode : BOOL;
    FeedStart_S4_UnLoad : BOOL;
    FeedFinish_S4_UnLoad : BOOL;
    FeedStart_S4_Load : BOOL;
    FeedFinish_S4_Load : BOOL;
    HMIPB_SOL_S4_UnLoad_PanelClip : BOOL;
    LS_S4_UnLoad_PanelUpDown1Out : BOOL;
    SOL_S4_UnLoad_PanelClip : BOOL;
    HMIPB_SOL_S4_Center_Clip : BOOL;
    SOL_S4_Center_Clip : BOOL;
    HMIPB_SOL_S4_Center_UpDown : BOOL;
    SOL_S4_Center_UpDown : BOOL;
    FeedStart : ARRAY[0..19] OF BOOL;
    FeedFinish : ARRAY[0..19] OF BOOL;
    HMIPB_S4_UnLoadGo : BOOL;
    HMIPB_S4_LoadGo : BOOL;
    LS_S4_Load_PanelUpDown1Back : BOOL;
    LS_S4_Load_PanelUpDown2Back : BOOL;
    LS_S4_UnLoad_PanelUpDown1Back : BOOL;
    LS_S4_UnLoad_PanelUpDown2Back : BOOL;
    HMISV_S4_Position : INT;
    HMIPB_S4_FeedTest : BOOL;
    ErrorStatus_S4_Center : BOOL;
END_VAR
(******************************************************************
程式:轉子送料
作者:Andy_Wang
版本資訊:1.0.0		2017/11/28
PowerOn=0
Idle=1
取料開始=2
夾取開=3
向上=4
移位至下一點=5
未到位門開啟設備暫停=20
StepMode解除=30
到位=6
向下=7
夾取出=8
向上=9
移位置放料=10
未到位門開啟設備暫停=21
StepMode解除=31
到位=11
向下=12
夾取歸=13
向上=14
移位置待機=15
未到位門開啟設備暫停=22
StepMode解除=32
到位=16
******************************************************************)
Error_LS:=ErrorStatus_S4_Center;
//PowerOn=0
IF NOT(SystemReadyStatus) OR Error_PB_EStop OR Error_LS THEN
	AutoFlow:=0;
END_IF;

//Idle=1
IF AutoFlow=0 AND NOT(Error_PB_EStop) AND  SystemReadyStatus  AND NOT(Error_LS)  THEN
	AutoFlow:=1;
END_IF;
IF AutoFlow=16 AND NOT(FeedFinish[4]) THEN
	AutoFlow:=1;
END_IF;
IF AutoFlow=1 THEN
	AutoFlow_Ready:=TRUE;
ELSE
	AutoFlow_Ready:=FALSE;
END_IF;

//取料開始=2
IF AutoFlow=1 AND
     (FeedStart[4] OR (HMIPB_S4_FeedTest AND NOT(AutoStatus)))AND 
	 HMISV_S4_Position<50 AND
	 AutoFlow2_Ready  and
	 AutoFlow2=1 THEN
	AutoFlow:=2;
END_IF;

//夾取開=3
IF AutoFlow=2  AND (Rtrig_test.Q OR NOT(StepMode)) THEN
	AutoFlow:=3;
  // load_Finish:=FALSE;
END_IF;

//向上=4
IF AutoFlow=3 AND
    LS_S4_Center_ClipBack AND
	//NOT(load_Finish) AND 
	(Rtrig_test.Q OR NOT(StepMode)) THEN
	AutoFlow:=4;
END_IF;

//移位至下一點=5
IF AutoFlow=4 AND LS_S4_Center_UpDownBack  AND (Rtrig_test.Q OR NOT(StepMode))  THEN
	AutoFlow:=5;
END_IF;

MC_MoveAbsolute_X_6(Axis:=MC_Axis000,  Execute:=AutoFlow=5 AND Ax_X.bServoOn AND MC_Axis000.Details.Homed
,  Position:=ServoS4_X_Table[ServoS4_X_Position,ServoS4_Y_Position],  Velocity:=HMISV_S4_AbsSpeedX, Acceleration:=5000,  Deceleration:=5000);
MC_MoveAbsolute_Y_6(Axis:=MC_Axis001, Execute:=AutoFlow=5 AND Ax_Y.bServoOn AND MC_Axis001.Details.Homed
, Position:=ServoS4_Y_Table[ServoS4_X_Position,ServoS4_Y_Position], Velocity:=HMISV_S4_AbsSpeedX, Acceleration:=5000, Deceleration:=5000);
 
 //未到位門開啟設備暫停=20
 IF AutoFlow=5 AND StepMode THEN
	 AutoFlow:=20;
 END_IF;
 //StepMode解除=30
 IF AutoFlow=20 AND NOT(StepMode) THEN
	 AutoFlow:=30;
 END_IF;
  IF AutoFlow=30 AND NOT(Ax_X.pbStop) AND NOT(Ax_Y.pbStop) THEN
	  AutoFlow:=5;
  END_IF;
 //到位=6
 IF AutoFlow=5  AND MC_MoveAbsolute_X_6.Done AND MC_MoveAbsolute_Y_6.Done  THEN
	 AutoFlow:=6;
 END_IF;
 
 //向下=7
 IF AutoFlow=6 AND (Rtrig_test.Q OR NOT(StepMode)) THEN
	 AutoFlow:=7;
 END_IF;
 
 //夾取出=8
 TON_1(In:=AutoFlow=7 AND LS_S4_Center_UpDownOut, PT:=t#300ms);
 IF AutoFlow=7 AND TON_1.Q AND (Rtrig_test.Q OR NOT(StepMode))  THEN
	 AutoFlow:=8;
 END_IF;
 
 //向上=9
  TON_2(In:=AutoFlow=8 AND LS_S4_Center_ClipOut, PT:=t#300ms);
  IF AutoFlow=8 AND TON_2.Q AND (Rtrig_test.Q OR NOT(StepMode)) THEN
	  AutoFlow:=9;
	  HMISV_S4_Position:=HMISV_S4_Position+1;
  END_IF;
 R_TRIG_1(Clk:=AutoFlow=9); 
(* IF  R_TRIG_1.Q AND  ServoS4_Y_Position<=9    THEN
	ServoS4_Y_Position:=ServoS4_Y_Position+1;
END_IF;*)
  
  //移位置放料=10
  IF AutoFlow=9 AND LS_S4_Center_UpDownBack AND (Rtrig_test.Q OR NOT(StepMode)) THEN
	  AutoFlow:=10;
  END_IF;
 
MC_MoveAbsolute_X_10(Axis:=MC_Axis001,  Execute:=AutoFlow=10 AND Ax_Y.bServoOn AND MC_Axis001.Details.Homed
,  Position:=ServoS4_PutPosition,  Velocity:=HMISV_S4_AbsSpeedX, Acceleration:=5000,  Deceleration:=5000);

(* R_TRIG_4(Clk:=AutoFlow=10); 
 IF R_TRIG_4.Q AND  ServoS4_Y_Position=10 AND ServoS4_X_Position<=4 THEN
	ServoS4_X_Position:=ServoS4_X_Position+1;
	ServoS4_Y_Position:=0;
END_IF; *)
  
//未到位門開啟設備暫停=21
IF AutoFlow=10 AND StepMode THEN
	AutoFlow:=21;
END_IF;
//StepMode解除=31
 IF AutoFlow=21 AND NOT(StepMode) THEN
	 AutoFlow:=31;
 END_IF;
  IF AutoFlow=31 AND NOT(Ax_X.pbStop) AND NOT(Ax_Y.pbStop) THEN
	  AutoFlow:=10;
  END_IF;
  
  //到位=11
  IF AutoFlow=10 AND MC_MoveAbsolute_X_10.Done AND (Rtrig_test.Q OR NOT(StepMode)) THEN
	  AutoFlow:=11;
  END_IF;
  
  //向下=12
  IF AutoFlow=11 AND (Rtrig_test.Q OR NOT(StepMode)) THEN 
	  AutoFlow:=12;
  END_IF;
  
  //夾取歸=13
  IF AutoFlow=12 AND LS_S4_Center_UpDownOut  AND (Rtrig_test.Q OR NOT(StepMode))  THEN
	  AutoFlow:=13;
  END_IF;
  
  //向上=14
  TON_3(In:=AutoFlow=13 AND LS_S4_Center_ClipBack, PT:=t#300ms);
  IF AutoFlow=13 AND TON_3.Q  AND (Rtrig_test.Q OR NOT(StepMode))  THEN
	  AutoFlow:=14;
  END_IF;
  
  //移位置待機=15
  IF AutoFlow=14 AND LS_S4_Center_UpDownBack  AND (Rtrig_test.Q OR NOT(StepMode))  THEN
	  AutoFlow:=15;
	    FeedFinish[4]:=TRUE;
  END_IF;
  MC_MoveAbsolute_X_15(Axis:=MC_Axis001,  Execute:=AutoFlow=15 AND Ax_Y.bServoOn AND MC_Axis001.Details.Homed
,  Position:=ServoS4_StandbyPosition,  Velocity:=HMISV_S4_AbsSpeedX, Acceleration:=5000,  Deceleration:=5000);
  
  //未到位門開啟設備暫停=22
IF AutoFlow=15 AND StepMode THEN
	AutoFlow:=22;
	  FeedFinish[4]:=FALSE;
END_IF;
//StepMode解除=32
 IF AutoFlow=22 AND NOT(StepMode) THEN
	 AutoFlow:=32;
 END_IF;
  IF AutoFlow=32 AND NOT(Ax_X.pbStop) AND NOT(Ax_Y.pbStop) THEN
	  AutoFlow:=15;
  END_IF;
  
  //到位=16
  IF AutoFlow=15 AND MC_MoveAbsolute_X_15.Done  THEN
	  AutoFlow:=16;
	   FeedFinish[4]:=FALSE;
  END_IF;
  (******************************************************************
程式:轉子收送盤
作者:Andy_Wang
版本資訊:1.0.0		2017/11/28
PowerOn=0
Idle=1 
   |-----------------------------------------------|
收盤開始=2                                            放盤開始=11
移至收盤位=3                                         移至放盤位=7
未到位門開啟設備暫停=20                   未到位門開啟設備暫停=21
StepMode解除=30									StepMode解除=31
到位=4                                                  到位=8
Call_Unload=5                                      Call_load=9
Unload_Finish=6                                   load_Finish=10
******************************************************************)
//PowerOn=0
IF NOT(SystemReadyStatus) OR Error_PB_EStop THEN
	AutoFlow2:=0;
END_IF;

//Idle=1
IF AutoFlow2=0 AND NOT(Error_PB_EStop) AND  SystemReadyStatus THEN
	AutoFlow2:=1;
END_IF;
IF AutoFlow2=6 AND NOT(AutoStatus) AND NOT(FeedStart_S4_UNLoad) AND Unload_Finish THEN
	AutoFlow2:=1;
END_IF;
IF AutoFlow2=10 AND NOT(FeedStart_S4_Load) AND load_Finish THEN
	AutoFlow2:=1;
END_IF;

IF AutoFlow2=1 THEN
	AutoFlow2_Ready:=TRUE;
ELSE
	AutoFlow2_Ready:=FALSE;
END_IF;
R_TRIG_5(CLK:=HMIPB_S4_UnLoadGo AND NOT(AutoStatus));
//收盤開始=2
IF  AutoFlow2=1 AND 
	 LS_S4_Center_UpDownBack AND	 NOT(SOL_S4_Center_UpDown) AND
	 LS_S4_Load_PanelUpDown1Back AND LS_S4_Load_PanelUpDown2Back AND LS_S4_UnLoad_PanelUpDown1Back AND LS_S4_UnLoad_PanelUpDown2Back AND
     ((ServoS4_Y_Position>=10 AND AutoStatus ) OR (R_TRIG_5.Q))   THEN
	AutoFlow2:=2;
END_IF;

//移至收盤位=3	
IF AutoFlow2=2 THEN
	AutoFlow2:=3;
	load_Finish:=FALSE;
	HMISV_S4_Position:=0;
END_IF;
  MC_MoveAbsolute_Y_3(Axis:=MC_Axis000,  Execute:=AutoFlow2=3 AND Ax_X.bServoOn AND MC_Axis000.Details.Homed
,  Position:=ServoS4_UnLoadPosition,  Velocity:=HMISV_S4_AbsSpeedX, Acceleration:=5000,  Deceleration:=5000);

//未到位門開啟設備暫停=20
IF AutoFlow2=3 AND StepMode  AND NOT(load_Finish) AND  ServoS4_X_Position =0 and ServoS4_Y_Position=0 THEN
	AutoFlow2:=20;
END_IF;
//StepMode解除=30
 IF AutoFlow2=20 AND NOT(StepMode) THEN
	 AutoFlow2:=30;
 END_IF;
  IF AutoFlow2=30 AND NOT(Ax_X.pbStop) THEN
	  AutoFlow2:=3;
  END_IF;

//到位=4
IF AutoFlow2=3 AND NOT(StepMode) AND MC_MoveAbsolute_Y_3.Done THEN
	AutoFlow2:=4;
END_IF;

//Call_Unload=5
IF AutoFlow2=4  THEN
	AutoFlow2:=5;
	FeedStart_S4_UnLoad:=TRUE;
END_IF;
IF FeedFinish_S4_UnLoad THEN
	FeedStart_S4_UnLoad:=FALSE;
END_IF;

//Unload_Finish=6
IF AutoFlow2=5 AND FeedFinish_S4_UnLoad THEN
	AutoFlow2:=6;
	Unload_Finish:=TRUE;
END_IF;

R_TRIG_6(CLK:=HMIPB_S4_LoadGo AND NOT(AutoStatus));
//放盤開始=11
IF  AutoFlow2=1 AND LS_S4_Center_UpDownBack AND NOT(SOL_S4_Center_UpDown) AND
	LS_S4_Load_PanelUpDown1Back AND LS_S4_Load_PanelUpDown2Back AND LS_S4_UnLoad_PanelUpDown1Back AND LS_S4_UnLoad_PanelUpDown2Back AND
	(R_TRIG_6.Q )  THEN
	AutoFlow2:=11;
	Unload_Finish:=FALSE;
END_IF;
IF AutoFlow2=6 AND (AutoStatus) AND NOT(FeedStart_S4_UNLoad) AND Unload_Finish THEN
	AutoFlow2:=11;
END_IF;

//移至放盤位=7
IF AutoFlow2=11 THEN
	AutoFlow2:=7;
END_IF;

 MC_MoveAbsolute_Y_7(Axis:=MC_Axis000,  Execute:=AutoFlow2=7 AND Ax_X.bServoOn AND MC_Axis000.Details.Homed
,  Position:=ServoS4_LoadPosition,  Velocity:=HMISV_S4_AbsSpeedX, Acceleration:=5000,  Deceleration:=5000);
 
//未到位門開啟設備暫停=21
IF AutoFlow2=7 AND StepMode THEN
	AutoFlow2:=21;
END_IF;
//StepMode解除=31
 IF AutoFlow2=21 AND NOT(StepMode) THEN
	 AutoFlow2:=31;
 END_IF;
  IF AutoFlow2=31 AND NOT(Ax_X.pbStop) THEN
	  AutoFlow2:=7;
  END_IF;
 
 //到位=8
IF AutoFlow2=7 AND MC_MoveAbsolute_Y_7.Done THEN
	AutoFlow2:=8;
END_IF;

//Call_load=9
IF AutoFlow2=8 THEN
	AutoFlow2:=9;
	FeedStart_S4_Load:=TRUE;
END_IF;
IF FeedFinish_S4_Load THEN
	FeedStart_S4_Load:=FALSE;
END_IF;
//load_Finish=10
IF AutoFlow2=9 AND NOT(FeedStart_S4_Load) AND ServoS4_X_Position=0 AND ServoS4_Y_Position=0 THEN
	AutoFlow2:=10;
	load_Finish:=TRUE;
END_IF;
//***************************************************************************************************************
(*取料夾取電磁閥*)
R_TRIG_2(CLK:=HMIPB_SOL_S4_Center_Clip AND NOT(AutoStatus));
interlockback[0]:=TRUE;
interlockout[0]:=TRUE;
(*SET*)
IF ((R_TRIG_2.Q AND NOT(solStatus[0])) OR Autoflow=8) AND interlockout[0] THEN
	SOL_S4_Center_Clip:=TRUE;
END_IF;
(*RESET*)
IF ((R_TRIG_2.Q AND (solStatus[0])) OR Autoflow=3 OR AutoFlow=13 OR Initflow=2) AND interlockback[0] THEN
	SOL_S4_Center_Clip:=FALSE;
END_IF;
(*STATUS*)
solStatus[0]:=SOL_S4_Center_Clip;
(*取料上下電磁閥*)
R_TRIG_3(CLK:=HMIPB_SOL_S4_Center_UpDown AND NOT(AutoStatus));
interlockback[1]:=TRUE;
interlockout[1]:=TRUE;
(*SET*)
IF ((R_TRIG_3.Q AND NOT(solStatus[1])) OR Autoflow=7 OR AutoFlow=12 ) AND interlockout[1] THEN
	SOL_S4_Center_UpDown:=TRUE;
END_IF;
(*RESET*)
IF ((R_TRIG_3.Q AND (solStatus[1])) OR Autoflow=4 OR AutoFlow=9  OR AutoFlow=14 OR Initflow=3) AND interlockback[1] THEN
	SOL_S4_Center_UpDown:=FALSE;
END_IF;
(*STATUS*)
solStatus[1]:=SOL_S4_Center_UpDown;
(**********************************************************************
程序名稱: 轉子送料 RESET程序
作者:Andy Wang
版本,日期,版本資訊:
1.0.0		2017/11/29		初始版本

PowerOn=0
Idle=1
夾取回=2
上下回=3
回待機點=4
到位=5
*******************************************************************)
//PowerOn=0
IF NOT(SystemReadyStatus) THEN
	Initflow:=0;
END_IF;

//Idle=1
IF Initflow=0 AND SystemReadyStatus THEN
	Initflow:=1;
END_IF;

IF Initflow=5 AND  LS_S4_Center_UpDownBack THEN
	Initflow:=1;
END_IF;

//夾取回=2
F_TRIG_1(Clk:=Error_LS);
IF Initflow=1 AND F_TRIG_1.Q THEN
	Initflow:=2;
END_IF;

//上下回=3
IF Initflow=2 AND LS_S4_Center_ClipBack THEN
	Initflow:=3;
END_IF;

//回待機點=4
IF Initflow=3 AND LS_S4_Center_UpDownBack THEN
	Initflow:=4;
END_IF;
MC_MoveAbsolute_X_5_init(Axis:=MC_Axis001,  Execute:=Initflow=4 AND Ax_Y.bServoOn AND MC_Axis001.Details.Homed
,  Position:=ServoS4_StandbyPosition,  Velocity:=HMISV_S4_AbsSpeedX, Acceleration:=5000,  Deceleration:=5000);

  //到位=5
  IF Initflow=4 AND MC_MoveAbsolute_X_5_init.Done THEN
	  Initflow:=5;
  END_IF;
	
END_PROGRAM

PROGRAM prStation4_Axis
VAR
    MC_Power_Ax1 : MC_Power;
    MC_Reset_Ax1 : MC_Reset;
    MC_Home_Ax1 : MC_Home;
    MC_Stop_Ax1 : MC_Stop;
    MC_MoveJog_Ax1 : MC_MoveJog;
    MC_MoveAbsolute_Ax1 : MC_MoveAbsolute;
    MC_Power_Ax2 : MC_Power;
    MC_Reset_Ax2 : MC_Reset;
    MC_Home_Ax2 : MC_Home;
    MC_Stop_Ax2 : MC_Stop;
    MC_MoveJog_Ax2 : MC_MoveJog;
    MC_MoveAbsolute_Ax2 : MC_MoveAbsolute;
    R_TRIG_1 : R_TRIG;
    MC_MoveAbsolute1 : ARRAY[0..3] OF MC_MoveAbsolute;
END_VAR
VAR_EXTERNAL CONSTANT
    MC_Axis000 : _sAXIS_REF;
END_VAR
VAR_EXTERNAL
    Error_PB_EStop : BOOL;
    Ax_Y : stAxis;
END_VAR
VAR_EXTERNAL CONSTANT
    MC_Axis001 : _sAXIS_REF;
END_VAR
VAR_EXTERNAL
    PB_Reset : BOOL;
    PB_EStop : BOOL;
    ServoS4_X_Table : ARRAY[0..4,0..9] OF LREAL;
    ServoS4_Y_Table : ARRAY[0..4,0..9] OF LREAL;
    ServoS4_PutPosition : LREAL;
    HMIPB_S4_SetPoint : BOOL;
    ServoS4_StandbyPosition : LREAL;
    HMIPB_ServoS4_PutPosition : BOOL;
    HMIPB_ServoS4_UnLoadPosition : BOOL;
    ServoS4_UnLoadPosition : LREAL;
    HMIPB_ServoS4_LoadPosition : BOOL;
    ServoS4_LoadPosition : LREAL;
    HMISV_S4_CurrentPositionX : LREAL;
    HMISV_S4_CurrentPositionY : LREAL;
    HMI_S4_State_Homed_MC : BOOL;
    HMI_S4_State_Homed_X : BOOL;
    HMI_S4_State_Homed_Y : BOOL;
    HMI_S4_State_HomeSerching_X : BOOL;
    HMI_S4_State_HomeSerching_Y : BOOL;
    HMI_S4_State_Homing_MC : BOOL;
    HMIPB_S4_ServoX_Back : BOOL;
    HMIPB_S4_ServoX_Out : BOOL;
    AutoStatus : BOOL;
    LS_S4_Center_UpDownBack : BOOL;
    SOL_S4_Center_UpDown : BOOL;
    HMIPB_S4_ServoY_Out : BOOL;
    HMIPB_S4_ServoY_Back : BOOL;
    HMISV_S4_ServoXJogSpeed : LREAL;
    HMISV_S4_ServoYJogSpeed : LREAL;
    HMIPB_S4_PostionGo : BOOL;
    ServoS4_X_Position : INT;
    HMIPB_S4_ServoOn_Y : BOOL;
    HMISV_S4_Position : INT;
    ServoS4_Y_Position : INT;
    HMISV_S4_AbsSpeedY : LREAL;
    HMISV_S4_AbsSpeedX : LREAL;
    Ax_X : stAxis;
    HMISV_ServoS4_X_Table : LREAL;
    HMISV_ServoS4_Y_Table : LREAL;
    StepMode : BOOL;
    HMIPB_S4_ServoOn_X : BOOL;
    LS_S4_Load_PanelUpDown1Back : BOOL;
    LS_S4_Load_PanelUpDown2Back : BOOL;
    SOL_S4_Load_PanelUpDown1Back : BOOL;
    SOL_S4_Load_PanelUpDown1Out : BOOL;
    SOL_S4_Load_PanelUpDown2Back : BOOL;
    SOL_S4_Load_PanelUpDown2Out : BOOL;
    SOL_S4_UnLoad_PanelUpDown1Back : BOOL;
    SOL_S4_UnLoad_PanelUpDown1Out : BOOL;
    SOL_S4_UnLoad_PanelUpDown2Back : BOOL;
    SOL_S4_UnLoad_PanelUpDown2Out : BOOL;
    HMIPB_PB_Reset : BOOL;
    HMIPB_ServoS4_StandbyPosition : BOOL;
    HMIState_NLS_X : BOOL;
    HMIState_PLS_X : BOOL;
    HMIState_HomeSW_X : BOOL;
    HMIState_NLS_Y : BOOL;
    HMIState_PLS_Y : BOOL;
    HMIState_HomeSW_Y : BOOL;
    HMIPB_ServoS4_PutPosition_MoveStart : BOOL;
    HMIPB_ServoS4_StandbyPosition_MoveStart : BOOL;
    HMIPB_ServoS4_UnLoadPosition_MoveStart : BOOL;
    HMIPB_ServoS4_LoadPosition_MoveStart : BOOL;
    LS_S4_UnLoad_PanelUpDown1Back : BOOL;
    LS_S4_UnLoad_PanelUpDown2Back : BOOL;
END_VAR
(*X軸*)
//Servo on
Ax_X.pbServoOn:=HMIPB_S4_ServoOn_X;
MC_Power_Ax1(Axis:=MC_Axis000, Enable:=Ax_X.pbServoOn AND NOT(Error_PB_EStop));
//Reset
MC_Reset_Ax1(Axis:=MC_Axis000, Execute:=Ax_X.pbReset);
//Home
MC_Home_Ax1(Axis:=MC_Axis000, Execute:=Ax_X.pbSerchHome AND Ax_X.bServoOn);
//STOP
MC_Stop_Ax1(Axis:=MC_Axis000, Execute:=Ax_X.pbStop);
//JOG
MC_MoveJog_Ax1(Axis:=MC_Axis000, PositiveEnable:=Ax_X.pbJOGForward , NegativeEnable:=Ax_X.pbJOGBackward , Velocity:=Ax_X.lrMoveJogVelocity,acceleration:=5000,deceleration:=5000);
//絕對定位
MC_MoveAbsolute_Ax1(Axis:=MC_Axis000, Execute:=Ax_X.pbMoveAbs AND Ax_X.bServoOn AND MC_Axis000.Details.Homed,
					Position:=Ax_X.lrMoveAbsAddData,	Velocity:=Ax_X.lrMoveAbsVelocity,acceleration:=5000,deceleration:=5000,
					Done=>Ax_X.bMoveAbsDone);
//定義
//Servo On
Ax_X.bServoOn:=MC_Axis000.DrvStatus.ServoOn;
//找HOME
Ax_X.bHoming:=MC_Axis000.Status.Homing;
//現在位置
Ax_X.lrCurrentPosition:=MC_Axis000.Act.Pos;
//反向極限
Ax_X.bNLS:=MC_Axis000.DrvStatus.N_OT;
HMIState_NLS_X:=Ax_X.bNLS;
//正向極限
Ax_X.bPLS:=MC_Axis000.DrvStatus.P_OT;
HMIState_PLS_X:=Ax_X.bPLS;
//原點訊號
Ax_X.bHomeSwitch:=MC_Axis000.DrvStatus.HomeSw;
HMIState_HomeSW_X:=Ax_X.bHomeSwitch;
//*********************************************************************************************************************************************************
(*Y軸*)
//Servo on
Ax_Y.pbServoOn:=HMIPB_S4_ServoOn_Y;
MC_Power_Ax2(Axis:=MC_Axis001, Enable:=Ax_Y.pbServoOn AND NOT(Error_PB_EStop));
//Reset
MC_Reset_Ax2(Axis:=MC_Axis001, Execute:=Ax_Y.pbReset);
//Home
MC_Home_Ax2(Axis:=MC_Axis001, Execute:=Ax_Y.pbSerchHome AND Ax_Y.bServoOn);
//STOP
MC_Stop_Ax2(Axis:=MC_Axis001, Execute:=Ax_Y.pbStop  );
//JOG
MC_MoveJog_Ax2(Axis:=MC_Axis001, PositiveEnable:=Ax_Y.pbJOGForward  , NegativeEnable:=Ax_Y.pbJOGBackward  , Velocity:=Ax_Y.lrMoveJogVelocity,acceleration:=5000,deceleration:=5000);
//絕對定位
MC_MoveAbsolute_Ax2(Axis:=MC_Axis001, Execute:=Ax_Y.pbMoveAbs AND Ax_Y.bServoOn AND MC_Axis001.Details.Homed,
					Position:=Ax_Y.lrMoveAbsAddData,	Velocity:=Ax_Y.lrMoveAbsVelocity,acceleration:=5000,deceleration:=5000,
					Done=>Ax_Y.bMoveAbsDone);

//定義
//Servo On
Ax_Y.bServoOn:=MC_Axis001.DrvStatus.ServoOn;
//找HOME
Ax_Y.bHoming:=MC_Axis001.Status.Homing;
//現在位置
Ax_Y.lrCurrentPosition:=MC_Axis001.Act.Pos;
//反向極限
Ax_Y.bNLS:=MC_Axis001.DrvStatus.N_OT;
HMIState_NLS_Y:=Ax_Y.bNLS;
//正向極限
Ax_Y.bPLS:=MC_Axis001.DrvStatus.P_OT;
HMIState_PLS_Y:=Ax_Y.bPLS;
//原點訊號
Ax_Y.bHomeSwitch:=MC_Axis001.DrvStatus.HomeSw;
HMIState_HomeSW_Y:=Ax_Y.bHomeSwitch;

//RESET
Ax_X.pbReset:=PB_Reset OR HMIPB_PB_Reset;
Ax_Y.pbReset:=PB_Reset OR HMIPB_PB_Reset;
//Stop
Ax_X.pbStop:=NOT(PB_EStop) OR StepMode ;
Ax_Y.pbStop:=NOT(PB_EStop) OR StepMode ;

//HMI原點復歸完成顯示
HMI_S4_State_Homed_X:=MC_Axis000.Details.Homed;//X軸復歸完成
HMI_S4_State_Homed_Y:=MC_Axis001.Details.Homed;//Y軸復歸完成
HMI_S4_State_HomeSerching_X:=Ax_X.bHoming;//X軸復歸中
HMI_S4_State_HomeSerching_Y:=Ax_Y.bHoming;//Y軸復歸中
HMI_S4_State_Homed_MC:=HMI_S4_State_Homed_X AND HMI_S4_State_Homed_Y AND NOT(HMI_S4_State_Homing_MC);//原點復歸完成
HMI_S4_State_Homing_MC:=HMI_S4_State_HomeSerching_X OR HMI_S4_State_HomeSerching_Y;//原點復歸中

//*********************************************************************************************************************************************************
//X伺服手動出
Ax_X.pbJOGForward:=
Ax_X.bServoOn AND
HMIPB_S4_ServoX_Out AND
NOT(AutoStatus) AND
LS_S4_Center_UpDownBack AND
NOT(SOL_S4_Center_UpDown) AND
LS_S4_Load_PanelUpDown1Back AND
LS_S4_Load_PanelUpDown2Back AND
NOT(SOL_S4_Load_PanelUpDown1Back) AND
NOT(SOL_S4_Load_PanelUpDown1Out) AND
NOT(SOL_S4_Load_PanelUpDown2Back) AND
NOT(SOL_S4_Load_PanelUpDown2Out) AND
NOT(SOL_S4_UnLoad_PanelUpDown1Back) AND
NOT(SOL_S4_UnLoad_PanelUpDown1Out) AND
NOT(SOL_S4_UnLoad_PanelUpDown2Back) AND
NOT(SOL_S4_UnLoad_PanelUpDown2Out);
//X伺服手動歸
Ax_X.pbJOGBackward:=
Ax_X.bServoOn AND
HMIPB_S4_ServoX_Back AND
NOT(AutoStatus) AND
LS_S4_Center_UpDownBack AND
NOT(SOL_S4_Center_UpDown) AND
LS_S4_Load_PanelUpDown1Back AND
LS_S4_Load_PanelUpDown2Back AND
NOT(SOL_S4_Load_PanelUpDown1Back) AND
NOT(SOL_S4_Load_PanelUpDown1Out) AND
NOT(SOL_S4_Load_PanelUpDown2Back) AND
NOT(SOL_S4_Load_PanelUpDown2Out) AND
NOT(SOL_S4_UnLoad_PanelUpDown1Back) AND
NOT(SOL_S4_UnLoad_PanelUpDown1Out) AND
NOT(SOL_S4_UnLoad_PanelUpDown2Back) AND
NOT(SOL_S4_UnLoad_PanelUpDown2Out);
//Y伺服手動出
Ax_Y.pbJOGForward:=
Ax_Y.bServoOn AND
HMIPB_S4_ServoY_Out AND
NOT(AutoStatus) AND
LS_S4_Center_UpDownBack AND
NOT(SOL_S4_Center_UpDown);
//Y伺服手動歸
Ax_Y.pbJOGBackward:=
Ax_Y.bServoOn AND
HMIPB_S4_ServoY_Back AND
NOT(AutoStatus) AND
LS_S4_Center_UpDownBack AND
NOT(SOL_S4_Center_UpDown);
//手動速度
Ax_X.lrMoveJogVelocity:=HMISV_S4_ServoXJogSpeed;
Ax_Y.lrMoveJogVelocity:=Ax_X.lrMoveJogVelocity;
//自動速度
Ax_X.lrMoveAbsVelocity:=HMISV_S4_AbsSpeedX;
Ax_Y.lrMoveAbsVelocity:=Ax_X.lrMoveAbsVelocity;
//*********************************************************************************************************************************************************
(*定位啟動控制*)
R_TRIG_1(Clk:=HMIPB_S4_PostionGo AND NOT(AutoStatus)  AND Ax_X.bServoOn AND Ax_Y.bServoOn AND MC_Axis000.Details.Homed AND MC_Axis001.Details.Homed );
IF NOT(AutoStatus) AND R_TRIG_1.Q THEN
//ServoS4_X_Position:=HMISV_S4_Position MOD 10;
//ServoS4_Y_Position:=HMISV_S4_Position/10;
Ax_X.lrMoveAbsAddData:=ServoS4_X_Table[ServoS4_X_Position,ServoS4_Y_Position];
Ax_Y.lrMoveAbsAddData:=ServoS4_Y_Table[ServoS4_X_Position,ServoS4_Y_Position];
Ax_X.lrMoveAbsVelocity:=HMISV_S4_AbsSpeedX;
Ax_Y.lrMoveAbsVelocity:=HMISV_S4_AbsSpeedX;
  IF (Ax_X.lrMoveAbsAddData=ServoS4_X_Table[ServoS4_X_Position,ServoS4_Y_Position] )AND (Ax_Y.lrMoveAbsAddData=ServoS4_Y_Table[ServoS4_X_Position,ServoS4_Y_Position] )THEN
	  Ax_X.pbMoveAbs:=TRUE;
	  Ax_Y.pbMoveAbs:=TRUE;
  END_IF;
END_IF;
//位置到達
IF Ax_X.bMoveAbsDone OR NOT(PB_EStop) OR Ax_X.pbStop THEN
	 Ax_X.pbMoveAbs:=FALSE;
END_IF;
IF Ax_Y.bMoveAbsDone OR NOT(PB_EStop) OR Ax_Y.pbStop THEN
	Ax_Y.pbMoveAbs:=FALSE;
END_IF;


//各點位置顯示
ServoS4_X_Position:=HMISV_S4_Position MOD 5;
ServoS4_Y_Position:=HMISV_S4_Position/5;
HMISV_ServoS4_X_Table:=ServoS4_X_Table[ServoS4_X_Position,ServoS4_Y_Position];
HMISV_ServoS4_Y_Table:=ServoS4_Y_Table[ServoS4_X_Position,ServoS4_Y_Position];

//現在位置HMI
HMISV_S4_CurrentPositionX:=Ax_X.lrCurrentPosition;
HMISV_S4_CurrentPositionY:=Ax_Y.lrCurrentPosition;

//各點位置寫入
IF HMIPB_S4_SetPoint THEN
ServoS4_X_Table[ServoS4_X_Position,ServoS4_Y_Position]:=Ax_X.lrCurrentPosition;
ServoS4_Y_Table[ServoS4_X_Position,ServoS4_Y_Position]:=Ax_Y.lrCurrentPosition;
END_IF;

//放料位置寫入
IF HMIPB_ServoS4_PutPosition THEN
ServoS4_PutPosition:=Ax_Y.lrCurrentPosition;
END_IF;
MC_MoveAbsolute1[0](Axis:=MC_Axis001, Execute:=HMIPB_ServoS4_PutPosition_MoveStart AND Ax_Y.bServoOn AND MC_Axis001.Details.Homed AND LS_S4_Center_UpDownBack AND NOT(SOL_S4_Center_UpDown),
					Position:=ServoS4_PutPosition,	Velocity:=Ax_Y.lrMoveAbsVelocity,acceleration:=5000,deceleration:=5000);
//待機位置寫入
IF HMIPB_ServoS4_StandbyPosition THEN
ServoS4_StandbyPosition:=Ax_Y.lrCurrentPosition;
END_IF;
MC_MoveAbsolute1[1](Axis:=MC_Axis001, Execute:=HMIPB_ServoS4_StandbyPosition_MoveStart AND Ax_Y.bServoOn AND MC_Axis001.Details.Homed AND LS_S4_Center_UpDownBack AND NOT(SOL_S4_Center_UpDown),
					Position:=ServoS4_StandbyPosition,	Velocity:=Ax_Y.lrMoveAbsVelocity,acceleration:=5000,deceleration:=5000);
//收盤位置寫入
IF HMIPB_ServoS4_UnLoadPosition THEN
	ServoS4_UnLoadPosition:=Ax_X.lrCurrentPosition;
END_IF;
MC_MoveAbsolute1[2](Axis:=MC_Axis000, Execute:=HMIPB_ServoS4_UnLoadPosition_MoveStart AND Ax_Y.bServoOn AND MC_Axis001.Details.Homed AND LS_S4_Center_UpDownBack AND NOT(SOL_S4_Center_UpDown AND LS_S4_Load_PanelUpDown1Back AND LS_S4_Load_PanelUpDown2Back AND LS_S4_UnLoad_PanelUpDown1Back AND LS_S4_UnLoad_PanelUpDown2Back),
					Position:=ServoS4_UnLoadPosition,	Velocity:=Ax_Y.lrMoveAbsVelocity,acceleration:=5000,deceleration:=5000);
//放盤位置寫入
IF HMIPB_ServoS4_LoadPosition THEN
	ServoS4_LoadPosition:=Ax_X.lrCurrentPosition;
END_IF;
MC_MoveAbsolute1[3](Axis:=MC_Axis000, Execute:=HMIPB_ServoS4_LoadPosition_MoveStart AND Ax_Y.bServoOn AND MC_Axis001.Details.Homed AND LS_S4_Center_UpDownBack AND NOT(SOL_S4_Center_UpDown AND LS_S4_Load_PanelUpDown1Back AND LS_S4_Load_PanelUpDown2Back AND LS_S4_UnLoad_PanelUpDown1Back AND LS_S4_UnLoad_PanelUpDown2Back),
					Position:=ServoS4_LoadPosition,	Velocity:=Ax_Y.lrMoveAbsVelocity,acceleration:=5000,deceleration:=5000);
END_PROGRAM

PROGRAM S4_AddDeviation
VAR
    i : INT;
    j : INT;
END_VAR
VAR_EXTERNAL
    ServoS4_X_Table : ARRAY[0..4,0..9] OF LREAL;
    ServoS4_Y_Table : ARRAY[0..4,0..9] OF LREAL;
    ServoS4_Y_Deviation : LREAL;
    ServoS4_X_Deviation : LREAL;
END_VAR
VAR_EXTERNAL CONSTANT
    HMIPB_S4_Deviation : BOOL;
END_VAR
IF HMIPB_S4_Deviation  THEN
FOR j:=0   TO 4 BY 1 DO
	FOR i:=0 TO 9 BY 1 DO
		ServoS4_X_Table[j,i]:=ServoS4_X_Table[0,0]-(ServoS4_X_Deviation*j);
   	    ServoS4_Y_Table[j,i]:=ServoS4_Y_Table[0,0]-(ServoS4_Y_Deviation*i);
	END_FOR;
END_FOR;
END_IF;
END_PROGRAM

PROGRAM S4_伺服原點復歸
VAR
    AutoFlow : INT;
    F_TRIG_1 : F_TRIG;
    R_TRIG_1 : R_TRIG;
    TON_1 : TON;
END_VAR
VAR_EXTERNAL
    SystemReadyStatus : BOOL;
    Error_PB_EStop : BOOL;
    HMI_S4_State_Homed_MC : BOOL;
    HMIPB_S4_Set_Homed : BOOL;
    Ax_X : stAxis;
    Ax_Y : stAxis;
END_VAR
VAR_EXTERNAL CONSTANT
    MC_Axis000 : _sAXIS_REF;
    MC_Axis001 : _sAXIS_REF;
END_VAR
VAR_EXTERNAL
    PB_ServoOn_X : BOOL;
    PB_ServoOn_Y : BOOL;
    SOL_S4_Center_Clip : BOOL;
    LS_S4_Center_ClipBack : BOOL;
    SOL_S4_Center_UpDown : BOOL;
    LS_S4_Center_UpDownBack : BOOL;
    AutoStatus : BOOL;
    HMIPB_S4_ServoOn_X : BOOL;
    HMIPB_S4_ServoOn_Y : BOOL;
END_VAR
(******************************************************************
程式:原點復歸
作者:Andy_Wang
版本資訊:1.0.0		2017/9/16
Power_ON=0
IDLE=1
全部狀態RESET=2
RESRT完成=3
伺服未回HOME=4
伺服Servo on=5
伺服Ready=6
夾取歸=7
上下回=8
伺服XY軸Serch Home開始=9
伺服XY軸Serch Home中=10
伺服XY軸Serch Home完成=11
伺服XY軸完成=12

******************************************************************)
//Power_ON=0
IF NOT(SystemReadyStatus) THEN
	AutoFlow:=0;
END_IF;

//IDLE=1
IF AutoFlow=0 AND SystemReadyStatus THEN
	AutoFlow:=1;
END_IF;

IF AutoFlow=12  THEN
	AutoFlow:=1;
END_IF;

//全部狀態RESET=2
//F_TRIG_1(Clk:= Error_PB_EStop  AND  NOT(HMI_S4_State_Homed_MC) );
R_TRIG_1(Clk:=HMIPB_S4_Set_Homed );
IF AutoFlow=1 AND (F_TRIG_1.Q  OR R_TRIG_1.Q) THEN
	AutoFlow:=2;
END_IF;
IF AutoFlow=2 THEN
	Ax_X.pbSerchHome:=FALSE;
	Ax_Y.pbSerchHome:=FALSE;
	Ax_X.pbMoveAbs:=FALSE;
	Ax_Y.pbMoveAbs:=FALSE;
	HMIPB_S4_Set_Homed:=FALSE;
END_IF;
//伺服未回HOME=3
IF AutoFlow=2 AND NOT(Ax_X.pbSerchHome)  AND NOT(Ax_Y.pbSerchHome)  
	                     AND NOT(Ax_X.pbMoveAbs) AND NOT(Ax_Y.pbMoveAbs) THEN
	AutoFlow:=3;
END_IF;

//伺服未回HOME=4
IF AutoFlow=3 AND  ((NOT(MC_Axis000.Details.Homed) AND NOT(MC_Axis001.Details.Homed)) OR
	                              (MC_Axis000.Details.Homed AND MC_Axis001.Details.Homed) OR
								  (MC_Axis000.Details.Homed AND NOT(MC_Axis001.Details.Homed)) OR
								  (NOT(MC_Axis000.Details.Homed) AND MC_Axis001.Details.Homed))  THEN
	AutoFlow:=4;
END_IF;

//伺服Servo on=5
IF AutoFlow=4 THEN
	AutoFlow:=5;
END_IF;
IF AutoFlow=5 THEN
	HMIPB_S4_ServoOn_X:=TRUE;
	HMIPB_S4_ServoOn_Y:=TRUE;
END_IF;

//伺服Ready=6
IF AutoFlow=5 AND Ax_X.bServoOn AND Ax_Y.bServoOn AND MC_Axis000.DrvStatus.Ready AND MC_Axis001.DrvStatus.Ready THEN
	AutoFlow:=6;
END_IF;

//夾取歸=7
IF AutoFlow=6 THEN
	AutoFlow:=7;
END_IF;
IF AutoFlow=7 THEN
	SOL_S4_Center_Clip:=FALSE;
END_IF;

//上下回=8
IF AutoFlow=7 AND LS_S4_Center_ClipBack THEN
	AutoFlow:=8;
END_IF;
IF AutoFlow=8 THEN
	SOL_S4_Center_UpDown:=FALSE;
END_IF;

//伺服XY軸Serch Home開始=9
TON_1(In:=AutoFlow=8 AND LS_S4_Center_UpDownBack, PT:=T#300ms);
IF AutoFlow=8 AND TON_1.Q THEN
	AutoFlow:=9;
END_IF;
IF AutoFlow=9 THEN
	Ax_X.pbSerchHome:=TRUE;
	Ax_Y.pbSerchHome:=TRUE;
END_IF;

//伺服XY軸Serch Home中=10
IF  AutoFlow=9 AND ((Ax_X.pbSerchHome OR Ax_X.bHoming OR MC_Axis000.Details.Homed )AND
                                     (Ax_Y.pbSerchHome  OR Ax_Y.bHoming OR MC_Axis001.Details.Homed))                             
									 THEN
	AutoFlow:=10;
END_IF;
IF AutoFlow=10 AND (Ax_X.bHoming  OR MC_Axis000.Details.Homed)  THEN
	Ax_X.pbSerchHome:=FALSE;
END_IF;
IF AutoFlow=10 AND (Ax_Y.bHoming OR MC_Axis001.Details.Homed)  THEN
	Ax_Y.pbSerchHome:=FALSE;
END_IF;

//伺服XY軸Serch Home完成=11
IF AutoFlow=10 AND MC_Axis001.Details.Homed AND MC_Axis000.Details.Homed 
	                       AND NOT(Ax_X.pbSerchHome) AND NOT(Ax_Y.pbSerchHome)   THEN
	AutoFlow:=11;
END_IF;

//伺服XY軸完成=12
IF AutoFlow=11 THEN
	AutoFlow:=12;
END_IF;
//******************************************************************
END_PROGRAM

PROGRAM File_R_W
VAR
    FileRead_Busy : BOOL;
    FileRead_Ini : BOOL;
    FileRead_Stage : UINT;
    FileRead_Index : UINT;
    FileRead_FileOpen : FileOpen;
    FileWrite_FileOpen : FileOpen;
    FileRead_FileClose : FileClose;
    FileWrite_FileClose : FileClose;
    FileRead_FileGet : FileGets;
    FileWrite_Fileput : FilePuts;
    FileRead_FileSeek : FileSeek;
    FileWrite_FileSeek : FileSeek;
    File_Name_All : STRING[30];
    FileRead_FID : DWORD;
    FileGet_String : STRING[256];
    i1 : UINT;
    FileGet_FindNum : UINT;
    FileWrite_Ini : BOOL;
    FileWrite_Busy : BOOL;
    FileWrite_Stage : UINT;
    FileWrite_Index : UINT;
    FileWrite_FID : DWORD;
    FilePut_String : STRING[256];
    Variable_A_String : STRING[30];
    Variable_B_String : STRING[30];
    Variable_C_String : STRING[30];
    Variable_D_String : STRING[30];
    Variable_E_String : STRING[30];
    Variable_F_String : STRING[30];
    Variable_G_String : STRING[30];
    Variable_H_String : STRING[30];
    Variable_I_String : STRING[30];
    R_TRIG1 : R_TRIG;
    nowtime : DATE_AND_TIME;
    sdnt : DATE_AND_TIME;
    pbsetdt : BOOL;
    nowtimeST : _sDT;
END_VAR
VAR_EXTERNAL
    File_Read_Tri : BOOL;
    SDCard_Ready : BOOL;
END_VAR
VAR_EXTERNAL CONSTANT
    _Card1Ready : BOOL;
END_VAR
VAR_EXTERNAL
    File_Name : STRING[30];
    File_Write_Tri : BOOL;
    Variable_A : ARRAY[0..9] OF REAL;
    Variable_B : ARRAY[0..9] OF REAL;
    Variable_C : ARRAY[0..9] OF REAL;
    Variable_D : ARRAY[0..9] OF REAL;
    Variable_E : ARRAY[0..9] OF REAL;
    Variable_F : ARRAY[0..9] OF REAL;
    Variable_G : ARRAY[0..9] OF REAL;
    Variable_H : ARRAY[0..9] OF REAL;
    Variable_I : ARRAY[0..9] OF REAL;
    Variable_Name : ARRAY[0..9] OF STRING[30];
    Error_BatchOK : BOOL;
    BatchOKCount : DINT;
    BatchNGCount : DINT;
    BatchTargetCount : DINT;
END_VAR
VAR_EXTERNAL CONSTANT
    _CurrentTime : DATE_AND_TIME;
END_VAR
(*****************************************************************************************************************************************************************************************************
 *此範例為使用SD Card 讀/寫 數值進入『.CSV檔』，將各變數數值儲存成『.CSV檔』有可於PC上檢視並且修改之特色。
 *
 *範例條件：可儲存 Variable_A ~ Variable_I，總共9個變數。
 *                   Variable_A ~ Variable_I儲存的數量不必相同。EX. Variable_A為999個元素的陣列，Variable_B為9999個元素的陣列。其它以此類推。
 *儲存格式範例：
 *------------------------------------------------------------------------------------------------------------------------------------------------------------------------------------------------------------
 *       Variable_A       │       Variable_B       │       Variable_C       │       Variable_D       │       Variable_E       │       Variable_F       │       Variable_G       │       Variable_H       │       Variable_I       │
 *------------------------------------------------------------------------------------------------------------------------------------------------------------------------------------------------------------
 *Variable_A.Value[0]│Variable_B.Value[0]│Variable_C.Value[0]│Variable_D.Value[0]│Variable_E.Value[0]│Variable_F.Value[0]│Variable_G.Value[0]│Variable_H.Value[0]│Variable_I.Value[0]│
 *------------------------------------------------------------------------------------------------------------------------------------------------------------------------------------------------------------
 *Variable_A.Value[1]│Variable_B.Value[1]│Variable_C.Value[1]│Variable_D.Value[1]│Variable_E.Value[1]│Variable_F.Value[1]│Variable_G.Value[1]│Variable_H.Value[1]│Variable_I.Value[1]│
 *------------------------------------------------------------------------------------------------------------------------------------------------------------------------------------------------------------
 *Variable_A.Value[2]│Variable_B.Value[2]│Variable_C.Value[2]│Variable_D.Value[2]│Variable_E.Value[2]│Variable_F.Value[2]│Variable_G.Value[2]│Variable_H.Value[2]│Variable_I.Value[2]│
 *------------------------------------------------------------------------------------------------------------------------------------------------------------------------------------------------------------
              ：                │              ：             │              ：             │              ：             │              ：             │              ：             │              ：             │              ：              │              ：            │
			  ：                │              ：             │              ：             │              ：             │              ：             │              ：             │              ：             │              ：              │              ：            │
 *------------------------------------------------------------------------------------------------------------------------------------------------------------------------------------------------------------
 * Variable_A.Value[?]│Variable_B.Value[?]│Variable_C.Value[?]│Variable_D.Value[?]│ Variable_E.Value[?]│Variable_F.Value[?]│Variable_G.Value[?]│ Variable_H.Value[?]│ Variable_I.Value[?]│
 *------------------------------------------------------------------------------------------------------------------------------------------------------------------------------------------------------------			  
 ******************************************************************************************************************************************************************************************************)
  Variable_Name[0]:='OK COUNT';
 Variable_Name[1]:='NG COUNT';
 Variable_Name[2]:='TARGET COUNT';
 //Variable_Name[3]:='TARGET COUNT';
SDCard_Ready := _Card1Ready;                                  // _Card1Ready為系統變數實際偵測NJ上是否有抓到插入的SD Card.
(*File_Name_All := CONCAT( File_Name , '.CSV');          //功能：結合File_Name(指定讀取檔名)與'.CSV'*)
//**********************************************************************************************************************************
//*   CSV檔案讀取程式                                                                                                                                                                    *
//**********************************************************************************************************************************
//File_Read_Tri 為 讀取CSV檔的『觸發BOOL變數』。                                   File_Write_Tri 為 寫入CSV檔的『觸發BOOL變數』。
//FileRead_Ini 為 讀取CSV檔程式：初始化程序執行中的旗標。                    FileWrite_Ini 為 寫入CSV檔程式：初始化程序執行中的旗標。
//FileRead_Busy 為 讀取CSV檔程式：讀取資料程序執行中的旗標。             FileWrite_Busy 為 寫入CSV檔程式：讀取資料程序執行中的旗標。 

IF (( File_Read_Tri = TRUE ) AND ( FileRead_Busy = FALSE) AND ( FileRead_Ini = FALSE) AND  ( FileWrite_Busy = FALSE) AND ( FileWrite_Ini = FALSE) AND (SDCard_Ready = TRUE) ) THEN
	FileRead_Ini := TRUE;
	FileRead_Busy := TRUE;
END_IF;

IF (FileRead_Ini = TRUE) THEN
	FileRead_FileOpen( Execute := FALSE);
	FileRead_FileSeek(Execute := FALSE);
	FileRead_FileGet(Execute := FALSE);
	FileRead_FileClose(Execute := FALSE);
	FileRead_Stage := UINT#1;
	FileRead_Index := UINT#0;
	FileRead_Ini := FALSE;
END_IF;

IF (FileRead_Busy = TRUE) THEN
	CASE FileRead_Stage OF
		1:
		    FileRead_FileOpen( Execute := TRUE , FileName := File_Name_All , Mode :=_READ_EXIST, FileID => FileRead_FID);
			
			IF (FileRead_FileOpen.Done = TRUE) THEN
				FileRead_Stage := 2;
			END_IF;
			IF (FileRead_FileOpen.Error = TRUE) THEN
				FileRead_Stage := 50;
			END_IF;
			
		2:
		    FileRead_FileSeek( Execute := TRUE , FileID := FileRead_FID , Offset := DINT#0 , Origin := _SEEK_SET );
			
			IF (FileRead_FileSeek.Done = TRUE) THEN
				FileRead_Stage := 3;
			END_IF;
			IF (FileRead_FileSeek.Error = TRUE) THEN
				FileRead_Stage := 50;
			END_IF;	
			
		3:
		    FileRead_FileGet(Execute := TRUE , FileID := FileRead_FID , TrimLF := TRUE );
			
			IF ( FileRead_FileGet.Done = TRUE) THEN
			    FileGet_String := FileRead_FileGet.Out;

				FOR i1:=0 TO UINT#8 BY UINT#1 DO                                                                       //For迴圈次數根據變數多寡決定，此範例讀取變數A~I共9個。
				    FileGet_FindNum := FIND(FileGet_String , ',');

(*-------------------------讀取Variable_A  ~  Variable_I的資料程序-------------------------*)						
						IF (FileRead_Index = 0) THEN                                                                           //讀取文件的第一行為Variable_A ~ Variable_I的名稱，第二行將數值丟入Variable_A~I。
							IF (FileGet_FindNum > 1 ) THEN                                                                      //判斷『,』的字元於字串變數中若為第一位則代表無值。
							    Variable_Name[i1] := MID(FileGet_String , FileGet_FindNum-1 , UINT#1);
							ELSIF (FileGet_FindNum = 1) THEN
								Variable_Name[i1] := '';
							ELSE
								Variable_Name[i1] := FileGet_String;
							END_IF;
							
						ELSE 
							
(*此判斷為Variable_A  ~  Variable_I 各種變數的陣列大小不同，因此若文件的列數大於Variable_A  ~  Variable_I 各種變數的陣列大小時
不管文件是否有給值皆不將數值丟入Variable_A  ~  Variable_I 。*)
							IF (FileGet_FindNum >1 ) THEN                                                                      //判斷『,』的字元於字串變數中若為第一位則代表無值。
								CASE i1 OF                                                                                                      //若讀取『,』數值大於1時，判斷為有數值。將字串帶入變數。
						            0: (*----------------------------------------讀取Variable_A的資料程序----------------------------------------*)
									   IF  (FileRead_Index <= 10 ) THEN
								            Variable_A[FileRead_Index-1] := STRING_TO_REAL(MID(FileGet_String , FileGet_FindNum-1 , UINT#1));
									   END_IF;
									1:(*----------------------------------------讀取Variable_B的資料程序----------------------------------------*)
										IF  (FileRead_Index <= 10 ) THEN
								            Variable_B[FileRead_Index-1] := STRING_TO_REAL(MID(FileGet_String , FileGet_FindNum-1 , UINT#1));
										END_IF;
									2:(*----------------------------------------讀取Variable_C的資料程序----------------------------------------*)
										 IF  (FileRead_Index <= 10 ) THEN
								            Variable_C[FileRead_Index-1] := STRING_TO_REAL(MID(FileGet_String , FileGet_FindNum-1 , UINT#1));
										END_IF;
									3:(*----------------------------------------讀取Variable_D的資料程序----------------------------------------*)
										IF  (FileRead_Index <= 10 ) THEN
								            Variable_D[FileRead_Index-1] := STRING_TO_REAL(MID(FileGet_String , FileGet_FindNum-1 , UINT#1));	
										END_IF;
									4:(*----------------------------------------讀取Variable_E的資料程序----------------------------------------*)
										IF  (FileRead_Index <= 10 ) THEN
								            Variable_E[FileRead_Index-1] := STRING_TO_REAL(MID(FileGet_String , FileGet_FindNum-1 , UINT#1));
										END_IF;
									5:(*----------------------------------------讀取Variable_F的資料程序----------------------------------------*)
										IF  (FileRead_Index <= 10) THEN
								            Variable_F[FileRead_Index-1] := STRING_TO_REAL(MID(FileGet_String , FileGet_FindNum-1 , UINT#1));
										END_IF;
									6:(*----------------------------------------讀取Variable_G的資料程序----------------------------------------*)
										IF  (FileRead_Index <= 10) THEN
								            Variable_G[FileRead_Index-1] := STRING_TO_REAL(MID(FileGet_String , FileGet_FindNum-1 , UINT#1));
										END_IF;
									7:(*----------------------------------------讀取Variable_H的資料程序----------------------------------------*)
										IF  (FileRead_Index <= 10 ) THEN
								            Variable_H[FileRead_Index-1] := STRING_TO_REAL(MID(FileGet_String , FileGet_FindNum-1 , UINT#1));	
										END_IF;
								END_CASE;
								
							ELSIF (FileGet_FindNum = 1) THEN								
								CASE i1 OF                                                                                                      //若讀取『,』數值等於1時，判斷為無數值。將0帶入變數。
						            0:(*----------------------------------------讀取Variable_A的資料程序----------------------------------------*)
									    IF  (FileRead_Index <= 10 ) THEN
								            Variable_A[FileRead_Index-1] := 0;
									    END_IF;
									1:(*----------------------------------------讀取Variable_B的資料程序----------------------------------------*)
									    IF  (FileRead_Index <= 10 ) THEN
								            Variable_B[FileRead_Index-1] := 0;
										END_IF;
									2:(*----------------------------------------讀取Variable_C的資料程序----------------------------------------*)
									    IF  (FileRead_Index <= 10 ) THEN
								            Variable_C[FileRead_Index-1] := 0;
										END_IF;
									3:(*----------------------------------------讀取Variable_D的資料程序----------------------------------------*)
									    IF  (FileRead_Index <= 10 ) THEN
								            Variable_D[FileRead_Index-1] := 0;	
										END_IF;
									4:(*----------------------------------------讀取Variable_E的資料程序----------------------------------------*)
									    IF  (FileRead_Index <= 10 ) THEN
								            Variable_E[FileRead_Index-1] := 0;
										END_IF;
									5:(*----------------------------------------讀取Variable_F的資料程序----------------------------------------*)
									    IF  (FileRead_Index <= 10 ) THEN
								            Variable_F[FileRead_Index-1] := 0;
										END_IF;
									6:(*----------------------------------------讀取Variable_G的資料程序----------------------------------------*)
									    IF  (FileRead_Index <= 10 ) THEN
								            Variable_G[FileRead_Index-1] := 0;
										END_IF;
									7:(*----------------------------------------讀取Variable_H的資料程序----------------------------------------*)
									    IF  (FileRead_Index <= 10 ) THEN
								            Variable_H[FileRead_Index-1] := 0;		
										END_IF;
								END_CASE;
							ELSE
								                                                                                                                       //若讀取『,』數值等於0時，判斷為最後一個變數的數值。								
									   (*----------------------------------------讀取Variable_I的資料程序----------------------------------------*)
										IF  (FileRead_Index <= 10 ) THEN
											IF (LEN( FileGet_String ) > 0) THEN
								                Variable_I[FileRead_Index-1] := STRING_TO_REAL(FileGet_String );
											ELSE
												 Variable_I[FileRead_Index-1] :=0;
											END_IF;
										END_IF;
								
							END_IF;
						END_IF;

					
					FileGet_String := DELETE(FileGet_String ,  FileGet_FindNum , UINT#1);
				END_FOR;
				
				FileRead_Index := FileRead_Index +1;
				
			    IF (FileRead_FileGet.EOF = FALSE) THEN
				    FileRead_FileGet(Execute := FALSE );
				ELSE
				    FileRead_Stage := 4;
				END_IF;
			END_IF;
			
			IF (FileRead_FileGet.Error = TRUE ) THEN
				 FileRead_Stage :=50;
			END_IF;
			
		4:
			FileRead_FileClose(Execute := TRUE , FileID := FileRead_FID );
			
			IF (FileRead_FileClose.Done = TRUE ) THEN
				 FileRead_Busy := FALSE;
			END_IF;
			IF (FileRead_FileClose.Error = TRUE ) THEN
				 FileRead_Stage :=50;
			END_IF;
			
		50:
		     FileRead_Busy := FALSE;
			 
	END_CASE;
END_IF;

//**********************************************************************************************************************************
//*   CSV檔案寫入程式                                                                                                                                                                    *
//**********************************************************************************************************************************
//File_Read_Tri 為 讀取CSV檔的『觸發BOOL變數』。                                   File_Write_Tri 為 寫入CSV檔的『觸發BOOL變數』。
//FileRead_Ini 為 讀取CSV檔程式：初始化程序執行中的旗標。                    FileWrite_Ini 為 寫入CSV檔程式：初始化程序執行中的旗標。
//FileRead_Busy 為 讀取CSV檔程式：讀取資料程序執行中的旗標。             FileWrite_Busy 為 寫入CSV檔程式：讀取資料程序執行中的旗標。 

IF (( File_Write_Tri = TRUE ) AND ( FileWrite_Busy = FALSE) AND ( FileWrite_Ini = FALSE) AND ( FileRead_Busy = FALSE) AND ( FileRead_Ini = FALSE) AND (SDCard_Ready = TRUE) ) THEN
	FileWrite_Ini := TRUE;
	FileWrite_Busy := TRUE;
END_IF;

IF (FileWrite_Ini = TRUE) THEN
	FileWrite_FileOpen( Execute := FALSE);
	FileWrite_FileSeek(Execute := FALSE);
	FileWrite_Fileput(Execute := FALSE);
	FileWrite_FileClose(Execute := FALSE);
	FileWrite_Stage := UINT#1;
	FileWrite_Index := UINT#0;
	FileWrite_Ini := FALSE;
END_IF;

IF (FileWrite_Busy = TRUE) THEN
	CASE FileWrite_Stage OF
		1:
		    FileWrite_FileOpen( Execute := TRUE , FileName := File_Name_All , Mode :=_RDWR_CREATE , FileID => FileWrite_FID);
			
			IF (FileWrite_FileOpen.Done = TRUE) THEN
				FileWrite_Stage := 2;
			END_IF;
			IF (FileWrite_FileOpen.Error = TRUE) THEN
				FileWrite_Stage := 50;
			END_IF;
			
		2:
		    FileWrite_FileSeek( Execute := TRUE , FileID := FileWrite_FID , Offset := DINT#0 , Origin := _SEEK_SET );
			
			IF (FileWrite_FileSeek.Done = TRUE) THEN
				FileWrite_Stage := 3;
			END_IF;
			IF (FileWrite_FileSeek.Error = TRUE) THEN
				FileWrite_Stage := 50;
			END_IF;		
			
